C07306=1192.829,186.350,-57.414,-177.869,6.477,148.554
C07307=1192.833,186.102,-57.391,-177.872,6.475,148.554
C07308=1192.838,185.853,-57.368,-177.874,6.474,148.554
C07309=1192.842,185.604,-57.345,-177.877,6.472,148.555
C07310=1192.846,185.355,-57.322,-177.880,6.470,148.555
C07311=1192.852,185.085,-57.297,-177.883,6.467,148.555
C07312=1192.857,184.815,-57.272,-177.885,6.466,148.556
C07313=1192.862,184.546,-57.247,-177.888,6.464,148.556
C07314=1192.867,184.276,-57.222,-177.891,6.462,148.556
C07315=1192.872,184.027,-57.199,-177.893,6.460,148.557
C07316=1192.876,183.779,-57.177,-177.896,6.458,148.557
C07317=1192.881,183.530,-57.153,-177.899,6.457,148.558
C07318=1192.885,183.281,-57.131,-177.901,6.455,148.558
C07319=1192.890,183.032,-57.108,-177.904,6.453,148.558
C07320=1192.894,182.783,-57.084,-177.907,6.451,148.559
C07321=1192.899,182.535,-57.062,-177.909,6.449,148.559
C07322=1192.904,182.285,-57.039,-177.912,6.448,148.559
C07323=1192.908,182.036,-57.017,-177.915,6.446,148.560
C07324=1192.913,181.787,-56.993,-177.917,6.444,148.560
C07325=1192.918,181.538,-56.971,-177.920,6.442,148.560
C07326=1192.922,181.290,-56.948,-177.923,6.440,148.561
C07327=1192.927,181.040,-56.925,-177.925,6.439,148.561
C07328=1192.931,180.791,-56.903,-177.928,6.437,148.561
C07329=1192.937,180.543,-56.880,-177.931,6.435,148.562
C07330=1192.941,180.294,-56.857,-177.933,6.433,148.562
C07331=1192.946,180.044,-56.834,-177.936,6.431,148.563
C07332=1192.950,179.796,-56.812,-177.939,6.430,148.563
C07333=1192.955,179.547,-56.789,-177.941,6.428,148.563
C07334=1192.959,179.298,-56.767,-177.944,6.426,148.564
C07335=1192.964,179.049,-56.743,-177.947,6.424,148.564
C07336=1192.969,178.800,-56.722,-177.949,6.422,148.564
C07337=1192.973,178.551,-56.698,-177.952,6.421,148.565
C07338=1192.978,178.302,-56.676,-177.955,6.419,148.565
C07339=1192.983,178.054,-56.653,-177.957,6.417,148.565
C07340=1192.987,177.804,-56.631,-177.960,6.415,148.566
C07341=1192.992,177.555,-56.608,-177.962,6.414,148.566
C07342=1192.997,177.307,-56.586,-177.965,6.412,148.567
C07343=1193.001,177.058,-56.563,-177.968,6.411,148.567
C07344=1193.006,176.808,-56.541,-177.970,6.409,148.567
C07345=1193.010,176.560,-56.518,-177.973,6.407,148.568
C07346=1193.015,176.311,-56.496,-177.976,6.405,148.568
C07347=1193.019,176.062,-56.473,-177.978,6.403,148.568
C07348=1193.025,175.813,-56.451,-177.981,6.402,148.569
C07349=1193.029,175.564,-56.428,-177.984,6.400,148.569
C07350=1193.033,175.315,-56.406,-177.986,6.398,148.569
C07351=1193.039,175.066,-56.384,-177.989,6.396,148.570
C07352=1193.043,174.817,-56.361,-177.992,6.395,148.570
C07353=1193.048,174.569,-56.339,-177.994,6.393,148.570
C07354=1193.053,174.319,-56.316,-177.997,6.391,148.571
C07355=1193.056,174.070,-56.294,-178.000,6.389,148.571
C07356=1193.061,173.822,-56.272,-178.002,6.387,148.572
C07357=1193.066,173.573,-56.249,-178.004,6.386,148.572
C07358=1193.071,173.324,-56.227,-178.007,6.385,148.572
C07359=1193.075,173.075,-56.205,-178.010,6.383,148.573
C07360=1193.080,172.825,-56.182,-178.012,6.381,148.573
C07361=1193.085,172.577,-56.160,-178.016,6.380,148.574
C07362=1193.089,172.328,-56.138,-178.018,6.378,148.574
C07363=1193.095,172.079,-56.116,-178.021,6.376,148.574
C07364=1193.099,171.830,-56.093,-178.024,6.374,148.575
C07365=1193.103,171.581,-56.071,-178.026,6.372,148.575
C07366=1193.108,171.332,-56.048,-178.029,6.371,148.575
C07367=1193.113,171.082,-56.026,-178.032,6.369,148.576
C07368=1193.118,170.834,-56.005,-178.034,6.368,148.576
C07369=1193.122,170.585,-55.982,-178.036,6.366,148.577
C07370=1193.127,170.336,-55.960,-178.039,6.364,148.577
C07371=1193.131,170.087,-55.938,-178.042,6.362,148.577
C07372=1193.136,169.838,-55.916,-178.044,6.361,148.578
C07373=1193.141,169.589,-55.894,-178.047,6.359,148.578
C07374=1193.145,169.341,-55.872,-178.050,6.357,148.578
C07375=1193.150,169.091,-55.849,-178.052,6.355,148.579
C07376=1193.155,168.842,-55.827,-178.055,6.354,148.579
C07377=1193.159,168.593,-55.805,-178.058,6.352,148.579
C07378=1193.164,168.344,-55.783,-178.060,6.351,148.580
C07379=1193.168,168.095,-55.761,-178.063,6.349,148.580
C07380=1193.174,167.846,-55.739,-178.066,6.348,148.581
C07381=1193.178,167.597,-55.717,-178.068,6.346,148.581
C07382=1193.183,167.348,-55.695,-178.071,6.344,148.582
C07383=1193.187,167.099,-55.673,-178.074,6.342,148.582
C07384=1193.192,166.850,-55.652,-178.076,6.340,148.582
C07385=1193.196,166.601,-55.629,-178.079,6.339,148.583
C07386=1193.201,166.353,-55.607,-178.081,6.338,148.583
C07387=1193.206,166.103,-55.585,-178.084,6.336,148.583
C07388=1193.211,165.854,-55.563,-178.087,6.334,148.584
C07389=1193.215,165.605,-55.541,-178.089,6.332,148.584
C07390=1193.220,165.356,-55.519,-178.092,6.331,148.585
C07391=1193.225,165.108,-55.498,-178.095,6.329,148.585
C07392=1193.230,164.858,-55.476,-178.098,6.327,148.585
C07393=1193.234,164.609,-55.454,-178.100,6.326,148.586
C07394=1193.239,164.360,-55.432,-178.102,6.325,148.586
C07395=1193.244,164.111,-55.411,-178.105,6.323,148.587
C07396=1193.248,163.862,-55.389,-178.108,6.321,148.587
C07397=1193.253,163.613,-55.367,-178.111,6.319,148.587
C07398=1193.258,163.365,-55.345,-178.113,6.317,148.588
C07399=1193.262,163.115,-55.323,-178.116,6.316,148.588
C07400=1193.267,162.867,-55.302,-178.119,6.314,148.588
C07401=1193.271,162.617,-55.280,-178.121,6.313,148.589
C07402=1193.276,162.368,-55.259,-178.124,6.311,148.589
C07403=1193.281,162.119,-55.237,-178.126,6.310,148.590
C07404=1193.285,161.870,-55.215,-178.129,6.308,148.590
C07405=1193.290,161.621,-55.193,-178.132,6.306,148.591
C07406=1193.294,161.372,-55.171,-178.135,6.304,148.591
C07407=1193.299,161.123,-55.149,-178.137,6.303,148.591
C07408=1193.304,160.874,-55.128,-178.139,6.302,148.592
C07409=1193.309,160.625,-55.106,-178.142,6.300,148.592
C07410=1193.314,160.376,-55.085,-178.145,6.298,148.593
C07411=1193.319,160.128,-55.063,-178.148,6.297,148.593
C07412=1193.323,159.878,-55.042,-178.150,6.295,148.593
C07413=1193.328,159.629,-55.020,-178.153,6.294,148.594
C07414=1193.333,159.380,-54.998,-178.155,6.292,148.594
C07415=1193.338,159.111,-54.976,-178.158,6.290,148.595
C07416=1193.343,158.842,-54.952,-178.161,6.289,148.595
C07417=1193.347,158.573,-54.929,-178.164,6.287,148.596
C07418=1193.353,158.304,-54.905,-178.166,6.285,148.596
C07419=1193.357,158.055,-54.883,-178.169,6.283,148.596
C07420=1193.362,157.805,-54.862,-178.172,6.282,148.597
C07421=1193.367,157.557,-54.841,-178.175,6.280,148.597
C07422=1193.371,157.308,-54.819,-178.178,6.278,148.598
C07423=1193.376,157.059,-54.798,-178.180,6.277,148.598
C07424=1193.381,156.810,-54.777,-178.182,6.276,148.598
C07425=1193.386,156.561,-54.756,-178.185,6.274,148.599
C07426=1193.390,156.311,-54.734,-178.188,6.272,148.599
C07427=1193.395,156.063,-54.712,-178.191,6.271,148.600
C07428=1193.400,155.813,-54.691,-178.194,6.269,148.600
C07429=1193.404,155.565,-54.670,-178.196,6.268,148.600
C07430=1193.409,155.315,-54.649,-178.198,6.266,148.601
C07431=1193.414,155.066,-54.627,-178.201,6.264,148.601
C07432=1193.419,154.817,-54.606,-178.204,6.263,148.602
C07433=1193.423,154.568,-54.584,-178.206,6.261,148.602
C07434=1193.428,154.319,-54.563,-178.209,6.260,148.603
C07435=1193.433,154.070,-54.542,-178.212,6.258,148.603
C07436=1193.438,153.821,-54.521,-178.214,6.257,148.603
C07437=1193.443,153.572,-54.499,-178.217,6.255,148.604
C07438=1193.447,153.323,-54.478,-178.219,6.254,148.604
C07439=1193.451,153.074,-54.457,-178.222,6.252,148.604
C07440=1193.457,152.825,-54.436,-178.225,6.251,148.605
C07441=1193.461,152.576,-54.414,-178.228,6.249,148.605
C07442=1193.465,152.327,-54.393,-178.230,6.247,148.606
C07443=1193.470,152.078,-54.372,-178.233,6.246,148.606
C07444=1193.475,151.829,-54.351,-178.235,6.244,148.607
C07445=1193.480,151.580,-54.330,-178.238,6.243,148.607
C07446=1193.485,151.331,-54.309,-178.241,6.241,148.608
C07447=1193.489,151.081,-54.287,-178.243,6.240,148.608
C07448=1193.494,150.832,-54.267,-178.246,6.239,148.608
C07449=1193.499,150.583,-54.245,-178.249,6.237,148.609
C07450=1193.504,150.334,-54.224,-178.251,6.235,148.609
C07451=1193.508,150.085,-54.204,-178.254,6.234,148.610
C07452=1193.513,149.837,-54.182,-178.256,6.233,148.610
C07453=1193.518,149.587,-54.161,-178.259,6.231,148.610
C07454=1193.522,149.338,-54.141,-178.262,6.229,148.611
C07455=1193.527,149.089,-54.119,-178.265,6.227,148.611
C07456=1193.532,148.840,-54.098,-178.267,6.227,148.612
C07457=1193.537,148.591,-54.077,-178.270,6.225,148.612
C07458=1193.542,148.342,-54.057,-178.273,6.223,148.613
C07459=1193.546,148.093,-54.035,-178.275,6.221,148.613
C07460=1193.550,147.843,-54.014,-178.277,6.220,148.613
C07461=1193.556,147.594,-53.993,-178.280,6.219,148.614
C07462=1193.560,147.345,-53.973,-178.283,6.217,148.614
C07463=1193.565,147.096,-53.951,-178.286,6.215,148.615
C07464=1193.569,146.848,-53.931,-178.288,6.214,148.615
C07465=1193.574,146.598,-53.910,-178.291,6.213,148.616
C07466=1193.579,146.349,-53.889,-178.294,6.211,148.616
C07467=1193.584,146.100,-53.868,-178.296,6.209,148.617
C07468=1193.589,145.851,-53.847,-178.299,6.209,148.617
C07469=1193.593,145.602,-53.826,-178.301,6.207,148.617
C07470=1193.598,145.353,-53.805,-178.304,6.205,148.618
C07471=1193.602,145.104,-53.785,-178.307,6.204,148.618
C07472=1193.608,144.854,-53.764,-178.309,6.203,148.619
C07473=1193.612,144.605,-53.743,-178.312,6.201,148.619
C07474=1193.617,144.356,-53.722,-178.315,6.199,148.619
C07475=1193.622,144.107,-53.702,-178.317,6.198,148.620
C07476=1193.627,143.858,-53.681,-178.320,6.197,148.620
C07477=1193.631,143.609,-53.661,-178.323,6.195,148.621
C07478=1193.636,143.360,-53.640,-178.325,6.193,148.621
C07479=1193.641,143.111,-53.619,-178.328,6.193,148.622
C07480=1193.645,142.862,-53.598,-178.331,6.191,148.622
C07481=1193.650,142.613,-53.577,-178.333,6.189,148.623
C07482=1193.655,142.364,-53.557,-178.335,6.188,148.623
C07483=1193.660,142.115,-53.536,-178.338,6.186,148.623
C07484=1193.664,141.866,-53.516,-178.341,6.185,148.624
C07485=1193.669,141.617,-53.495,-178.344,6.183,148.624
C07486=1193.674,141.368,-53.474,-178.346,6.182,148.625
C07487=1193.679,141.118,-53.455,-178.349,6.180,148.625
C07488=1193.684,140.869,-53.434,-178.352,6.179,148.626
C07489=1193.688,140.620,-53.413,-178.354,6.178,148.626
C07490=1193.693,140.371,-53.393,-178.357,6.176,148.627
C07491=1193.698,140.122,-53.372,-178.359,6.174,148.627
C07492=1193.702,139.873,-53.351,-178.362,6.174,148.628
C07493=1193.707,139.624,-53.331,-178.365,6.172,148.628
C07494=1193.712,139.375,-53.310,-178.367,6.170,148.628
C07495=1193.716,139.126,-53.290,-178.370,6.169,148.629
C07496=1193.721,138.876,-53.269,-178.373,6.168,148.629
C07497=1193.726,138.627,-53.248,-178.375,6.166,148.630
C07498=1193.731,138.378,-53.229,-178.378,6.164,148.630
C07499=1193.736,138.129,-53.208,-178.381,6.164,148.631
C07500=1193.740,137.880,-53.187,-178.383,6.162,148.631
C07501=1193.745,137.631,-53.167,-178.386,6.160,148.632
C07502=1193.749,137.382,-53.147,-178.388,6.159,148.632
C07503=1193.755,137.132,-53.126,-178.391,6.158,148.633
C07504=1193.759,136.883,-53.106,-178.394,6.156,148.633
C07505=1193.763,136.634,-53.086,-178.396,6.155,148.633
C07506=1193.769,136.385,-53.065,-178.399,6.153,148.634
C07507=1193.773,136.135,-53.045,-178.402,6.152,148.634
C07508=1193.778,135.886,-53.025,-178.404,6.151,148.635
C07509=1193.782,135.637,-53.004,-178.407,6.149,148.635
C07510=1193.788,135.389,-52.984,-178.410,6.148,148.636
C07511=1193.793,135.139,-52.964,-178.412,6.147,148.636
C07512=1193.797,134.890,-52.944,-178.415,6.145,148.637
C07513=1193.802,134.641,-52.923,-178.417,6.143,148.637
C07514=1193.806,134.392,-52.904,-178.420,6.143,148.638
C07515=1193.812,134.142,-52.883,-178.423,6.141,148.638
C07516=1193.816,133.893,-52.862,-178.425,6.139,148.638
C07517=1193.821,133.644,-52.843,-178.428,6.139,148.639
C07518=1193.825,133.395,-52.822,-178.431,6.137,148.639
C07519=1193.831,133.127,-52.800,-178.433,6.135,148.640
C07520=1193.835,132.858,-52.779,-178.437,6.134,148.640
C07521=1193.841,132.589,-52.757,-178.439,6.132,148.641
C07522=1193.846,132.321,-52.735,-178.442,6.131,148.641
C07523=1193.851,132.071,-52.715,-178.445,6.130,148.642
C07524=1193.856,131.823,-52.695,-178.447,6.128,148.642
C07525=1193.861,131.573,-52.675,-178.450,6.127,148.643
C07526=1193.865,131.324,-52.655,-178.453,6.125,148.643
C07527=1193.870,131.075,-52.635,-178.455,6.124,148.644
C07528=1193.875,130.826,-52.615,-178.458,6.123,148.644
C07529=1193.879,130.577,-52.595,-178.461,6.121,148.645
C07530=1193.884,130.328,-52.575,-178.463,6.120,148.645
C07531=1193.890,130.079,-52.554,-178.465,6.119,148.645
C07532=1193.894,129.829,-52.535,-178.469,6.117,148.646
C07533=1193.899,129.580,-52.514,-178.471,6.115,148.646
C07534=1193.903,129.331,-52.495,-178.473,6.114,148.647
C07535=1193.909,129.082,-52.475,-178.476,6.113,148.647
C07536=1193.913,128.833,-52.455,-178.479,6.112,148.648
C07537=1193.918,128.583,-52.435,-178.481,6.110,148.648
C07538=1193.922,128.334,-52.415,-178.484,6.109,148.649
C07539=1193.927,128.085,-52.395,-178.487,6.108,148.649
C07540=1193.932,127.837,-52.375,-178.489,6.106,148.650
C07541=1193.937,127.587,-52.356,-178.492,6.106,148.650
C07542=1193.941,127.338,-52.335,-178.495,6.104,148.651
C07543=1193.946,127.088,-52.316,-178.497,6.102,148.651
C07544=1193.951,126.840,-52.296,-178.500,6.102,148.652
C07545=1193.956,126.591,-52.276,-178.503,6.100,148.652
C07546=1193.961,126.341,-52.256,-178.505,6.098,148.652
C07547=1193.965,126.091,-52.237,-178.508,6.097,148.653
C07548=1193.970,125.843,-52.217,-178.511,6.096,148.653
C07549=1193.975,125.594,-52.197,-178.513,6.095,148.654
C07550=1193.980,125.344,-52.177,-178.516,6.093,148.654
C07551=1193.984,125.095,-52.157,-178.519,6.092,148.655
C07552=1193.990,124.846,-52.138,-178.521,6.091,148.655
C07553=1193.994,124.597,-52.118,-178.524,6.089,148.656
C07554=1193.999,124.347,-52.098,-178.526,6.088,148.656
C07555=1194.004,124.098,-52.078,-178.529,6.087,148.657
C07556=1194.009,123.849,-52.059,-178.532,6.085,148.657
C07557=1194.013,123.600,-52.040,-178.534,6.084,148.658
C07558=1194.018,123.350,-52.020,-178.537,6.082,148.658
C07559=1194.023,123.102,-52.000,-178.539,6.082,148.659
C07560=1194.028,122.853,-51.980,-178.542,6.080,148.659
C07561=1194.032,122.603,-51.961,-178.544,6.079,148.660
C07562=1194.038,122.354,-51.941,-178.547,6.078,148.660
C07563=1194.042,122.105,-51.921,-178.550,6.076,148.661
C07564=1194.047,121.856,-51.901,-178.553,6.075,148.661
C07565=1194.052,121.607,-51.882,-178.555,6.074,148.662
C07566=1194.056,121.358,-51.863,-178.557,6.073,148.662
C07567=1194.061,121.108,-51.843,-178.561,6.071,148.663
C07568=1194.066,120.859,-51.824,-178.563,6.070,148.663
C07569=1194.071,120.610,-51.804,-178.565,6.069,148.663
C07570=1194.075,120.361,-51.784,-178.569,6.067,148.664
C07571=1194.081,120.112,-51.765,-178.571,6.066,148.664
C07572=1194.085,119.863,-51.746,-178.573,6.064,148.665
C07573=1194.089,119.613,-51.726,-178.576,6.064,148.666
C07574=1194.095,119.364,-51.707,-178.579,6.062,148.666
C07575=1194.100,119.115,-51.687,-178.582,6.061,148.667
C07576=1194.105,118.866,-51.668,-178.584,6.060,148.667
C07577=1194.109,118.616,-51.649,-178.587,6.058,148.667
C07578=1194.114,118.367,-51.629,-178.589,6.057,148.668
C07579=1194.119,118.118,-51.610,-178.592,6.056,148.668
C07580=1194.124,117.868,-51.590,-178.594,6.055,148.669
C07581=1194.128,117.620,-51.571,-178.597,6.053,148.669
C07582=1194.133,117.370,-51.552,-178.599,6.052,148.670
C07583=1194.138,117.121,-51.532,-178.603,6.051,148.670
C07584=1194.143,116.872,-51.513,-178.605,6.049,148.671
C07585=1194.147,116.623,-51.494,-178.607,6.048,148.671
C07586=1194.153,116.374,-51.475,-178.611,6.047,148.672
C07587=1194.157,116.124,-51.455,-178.613,6.046,148.672
C07588=1194.162,115.876,-51.436,-178.616,6.045,148.673
C07589=1194.167,115.626,-51.416,-178.618,6.044,148.673
C07590=1194.172,115.377,-51.397,-178.621,6.042,148.674
C07591=1194.177,115.128,-51.378,-178.623,6.041,148.674
C07592=1194.181,114.878,-51.358,-178.626,6.040,148.675
C07593=1194.186,114.629,-51.340,-178.629,6.039,148.675
C07594=1194.191,114.379,-51.320,-178.631,6.037,148.676
C07595=1194.196,114.131,-51.302,-178.634,6.036,148.676
C07596=1194.200,113.881,-51.282,-178.637,6.035,148.677
C07597=1194.206,113.632,-51.263,-178.639,6.034,148.677
C07598=1194.210,113.383,-51.244,-178.642,6.033,148.678
C07599=1194.215,113.134,-51.224,-178.645,6.031,148.678
C07600=1194.219,112.884,-51.206,-178.647,6.030,148.679
C07601=1194.225,112.635,-51.187,-178.650,6.029,148.679
C07602=1194.230,112.386,-51.167,-178.652,6.028,148.680
C07603=1194.234,112.137,-51.148,-178.655,6.026,148.680
C07604=1194.239,111.888,-51.129,-178.658,6.025,148.681
C07605=1194.244,111.639,-51.111,-178.660,6.023,148.681
C07606=1194.249,111.389,-51.091,-178.663,6.023,148.682
C07607=1194.254,111.140,-51.072,-178.666,6.021,148.682
C07608=1194.258,110.891,-51.053,-178.668,6.021,148.683
C07609=1194.264,110.641,-51.034,-178.671,6.019,148.683
C07610=1194.268,110.392,-51.015,-178.673,6.018,148.684
C07611=1194.273,110.143,-50.996,-178.676,6.017,148.684
C07612=1194.277,109.893,-50.977,-178.678,6.016,148.685
C07613=1194.283,109.645,-50.958,-178.681,6.014,148.685
C07614=1194.287,109.396,-50.939,-178.684,6.013,148.686
C07615=1194.292,109.146,-50.920,-178.687,6.012,148.686
C07616=1194.297,108.897,-50.902,-178.689,6.011,148.687
C07617=1194.302,108.648,-50.882,-178.692,6.010,148.687
C07618=1194.306,108.398,-50.864,-178.694,6.009,148.688
C07619=1194.311,108.149,-50.844,-178.697,6.007,148.688
C07620=1194.316,107.900,-50.826,-178.700,6.006,148.689
C07621=1194.321,107.650,-50.807,-178.702,6.005,148.689
C07622=1194.325,107.402,-50.788,-178.705,6.004,148.690
C07623=1194.331,107.133,-50.768,-178.708,6.002,148.690
C07624=1194.336,106.864,-50.747,-178.711,6.001,148.691
C07625=1194.341,106.596,-50.728,-178.713,6.000,148.692
C07626=1194.347,106.328,-50.707,-178.716,5.998,148.692
C07627=1194.351,106.078,-50.689,-178.719,5.998,148.693
C07628=1194.356,105.829,-50.669,-178.721,5.996,148.693
C07629=1194.361,105.580,-50.651,-178.724,5.996,148.694
C07630=1194.366,105.331,-50.632,-178.727,5.994,148.694
C07631=1194.371,105.082,-50.614,-178.729,5.993,148.695
C07632=1194.376,104.832,-50.594,-178.732,5.992,148.695
C07633=1194.381,104.583,-50.576,-178.734,5.991,148.696
C07634=1194.385,104.334,-50.557,-178.737,5.989,148.696
C07635=1194.390,104.084,-50.538,-178.739,5.988,148.697
C07636=1194.395,103.835,-50.520,-178.743,5.987,148.697
C07637=1194.400,103.586,-50.502,-178.745,5.986,148.698
C07638=1194.405,103.337,-50.482,-178.748,5.985,148.698
C07639=1194.410,103.088,-50.464,-178.750,5.984,148.699
C07640=1194.415,102.839,-50.445,-178.753,5.983,148.699
C07641=1194.419,102.589,-50.426,-178.755,5.981,148.700
C07642=1194.424,102.340,-50.408,-178.758,5.980,148.700
C07643=1194.429,102.091,-50.389,-178.761,5.979,148.701
C07644=1194.434,101.841,-50.371,-178.763,5.978,148.701
C07645=1194.438,101.592,-50.352,-178.766,5.977,148.702
C07646=1194.444,101.343,-50.334,-178.768,5.976,148.702
C07647=1194.448,101.093,-50.315,-178.771,5.974,148.703
C07648=1194.453,100.844,-50.296,-178.774,5.973,148.703
C07649=1194.458,100.595,-50.279,-178.777,5.972,148.704
C07650=1194.463,100.345,-50.260,-178.779,5.971,148.704
C07651=1194.467,100.096,-50.241,-178.781,5.971,148.705
C07652=1194.472,99.847,-50.223,-178.784,5.969,148.706
C07653=1194.477,99.597,-50.204,-178.787,5.968,148.706
C07654=1194.482,99.349,-50.185,-178.790,5.967,148.707
C07655=1194.487,99.099,-50.167,-178.792,5.966,148.707
C07656=1194.492,98.850,-50.149,-178.795,5.964,148.708
C07657=1194.497,98.600,-50.130,-178.797,5.964,148.708
C07658=1194.502,98.351,-50.112,-178.800,5.963,148.709
C07659=1194.506,98.102,-50.094,-178.803,5.961,148.709
C07660=1194.511,97.853,-50.076,-178.805,5.960,148.710
C07661=1194.516,97.603,-50.057,-178.808,5.959,148.710
C07662=1194.521,97.354,-50.039,-178.810,5.958,148.711
C07663=1194.526,97.105,-50.020,-178.813,5.957,148.711
C07664=1194.531,96.856,-50.002,-178.816,5.956,148.712
C07665=1194.535,96.606,-49.984,-178.818,5.955,148.713
C07666=1194.540,96.357,-49.966,-178.821,5.953,148.713
C07667=1194.546,96.107,-49.947,-178.824,5.953,148.714
C07668=1194.550,95.859,-49.929,-178.826,5.951,148.714
C07669=1194.555,95.610,-49.911,-178.829,5.951,148.715
C07670=1194.560,95.360,-49.892,-178.832,5.949,148.715
C07671=1194.564,95.111,-49.874,-178.834,5.948,148.716
C07672=1194.569,94.862,-49.856,-178.836,5.947,148.716
C07673=1194.574,94.612,-49.838,-178.840,5.946,148.717
C07674=1194.580,94.363,-49.820,-178.842,5.945,148.717
C07675=1194.584,94.113,-49.801,-178.845,5.944,148.718
C07676=1194.589,93.864,-49.783,-178.847,5.943,148.718
C07677=1194.594,93.615,-49.765,-178.850,5.942,148.719
C07678=1194.599,93.366,-49.747,-178.852,5.940,148.719
C07679=1194.604,93.117,-49.729,-178.855,5.940,148.720
C07680=1194.608,92.867,-49.710,-178.858,5.938,148.720
C07681=1194.613,92.618,-49.692,-178.860,5.938,148.721
C07682=1194.618,92.369,-49.674,-178.862,5.937,148.721
C07683=1194.623,92.120,-49.656,-178.866,5.935,148.722
C07684=1194.628,91.870,-49.638,-178.868,5.934,148.722
C07685=1194.633,91.621,-49.620,-178.871,5.933,148.723
C07686=1194.638,91.372,-49.602,-178.873,5.932,148.724
C07687=1194.642,91.122,-49.584,-178.876,5.932,148.724
C07688=1194.647,90.873,-49.566,-178.878,5.930,148.725
C07689=1194.652,90.623,-49.548,-178.881,5.929,148.725
C07690=1194.657,90.374,-49.530,-178.884,5.928,148.726
C07691=1194.662,90.125,-49.512,-178.886,5.927,148.726
C07692=1194.667,89.875,-49.494,-178.888,5.926,148.727
C07693=1194.672,89.626,-49.476,-178.892,5.925,148.727
C07694=1194.677,89.377,-49.458,-178.894,5.924,148.728
C07695=1194.681,89.127,-49.440,-178.896,5.923,148.728
C07696=1194.686,88.878,-49.422,-178.899,5.921,148.729
C07697=1194.691,88.629,-49.404,-178.902,5.921,148.730
C07698=1194.696,88.380,-49.386,-178.904,5.919,148.730
C07699=1194.701,88.130,-49.368,-178.907,5.919,148.731
C07700=1194.706,87.881,-49.350,-178.910,5.918,148.731
C07701=1194.711,87.631,-49.333,-178.912,5.916,148.732
C07702=1194.715,87.383,-49.315,-178.915,5.916,148.732
C07703=1194.720,87.133,-49.298,-178.917,5.915,148.733
C07704=1194.725,86.884,-49.280,-178.920,5.913,148.733
C07705=1194.730,86.635,-49.262,-178.923,5.913,148.734
C07706=1194.735,86.385,-49.244,-178.925,5.912,148.734
C07707=1194.740,86.136,-49.226,-178.928,5.910,148.735
C07708=1194.745,85.886,-49.208,-178.930,5.910,148.736
C07709=1194.749,85.637,-49.190,-178.933,5.908,148.736
C07710=1194.754,85.388,-49.172,-178.936,5.907,148.737
C07711=1194.760,85.138,-49.155,-178.938,5.907,148.737
C07712=1194.764,84.889,-49.137,-178.941,5.905,148.738
C07713=1194.769,84.640,-49.119,-178.944,5.905,148.738
C07714=1194.774,84.391,-49.101,-178.946,5.904,148.739
C07715=1194.779,84.141,-49.084,-178.949,5.902,148.739
C07716=1194.784,83.892,-49.066,-178.951,5.901,148.740
C07717=1194.789,83.643,-49.048,-178.954,5.901,148.740
C07718=1194.794,83.393,-49.031,-178.957,5.899,148.741
C07719=1194.799,83.144,-49.013,-178.959,5.898,148.742
C07720=1194.803,82.895,-48.996,-178.961,5.898,148.742
C07721=1194.808,82.645,-48.978,-178.965,5.896,148.743
C07722=1194.813,82.396,-48.960,-178.967,5.896,148.743
C07723=1194.818,82.147,-48.942,-178.969,5.895,148.744
C07724=1194.823,81.897,-48.925,-178.973,5.893,148.744
C07725=1194.827,81.648,-48.908,-178.975,5.892,148.745
C07726=1194.833,81.398,-48.890,-178.977,5.892,148.745
C07727=1194.838,81.130,-48.871,-178.980,5.891,148.746
C07728=1194.844,80.862,-48.853,-178.983,5.890,148.747
C07729=1194.849,80.594,-48.833,-178.986,5.888,148.747
C07730=1194.854,80.325,-48.815,-178.988,5.888,148.748
C07731=1194.858,80.076,-48.797,-178.991,5.886,148.748
C07732=1194.863,79.826,-48.780,-178.994,5.885,148.749
C07733=1194.868,79.577,-48.762,-178.996,5.885,148.750
C07734=1194.873,79.328,-48.744,-178.999,5.883,148.750
C07735=1194.878,79.078,-48.727,-179.002,5.883,148.751
C07736=1194.883,78.829,-48.709,-179.004,5.882,148.751
C07737=1194.889,78.580,-48.692,-179.007,5.880,148.752
C07738=1194.893,78.331,-48.674,-179.010,5.880,148.752
C07739=1194.898,78.081,-48.658,-179.012,5.879,148.753
C07740=1194.903,77.832,-48.640,-179.015,5.877,148.753
C07741=1194.908,77.582,-48.623,-179.017,5.877,148.754
C07742=1194.913,77.333,-48.606,-179.020,5.876,148.755
C07743=1194.917,77.084,-48.588,-179.022,5.875,148.755
C07744=1194.923,76.834,-48.571,-179.025,5.874,148.756
C07745=1194.927,76.585,-48.553,-179.028,5.873,148.756
C07746=1194.932,76.335,-48.536,-179.030,5.872,148.757
C07747=1194.937,76.086,-48.518,-179.033,5.871,148.757
C07748=1194.942,75.837,-48.502,-179.035,5.870,148.758
C07749=1194.947,75.587,-48.484,-179.038,5.869,148.758
C07750=1194.952,75.338,-48.466,-179.041,5.868,148.759
C07751=1194.957,75.089,-48.450,-179.043,5.867,148.760
C07752=1194.962,74.840,-48.432,-179.046,5.867,148.760
C07753=1194.966,74.590,-48.415,-179.048,5.866,148.761
C07754=1194.971,74.340,-48.398,-179.051,5.864,148.761
C07755=1194.977,74.092,-48.380,-179.053,5.863,148.762
C07756=1194.981,73.842,-48.364,-179.056,5.863,148.762
C07757=1194.986,73.593,-48.346,-179.059,5.862,148.763
C07758=1194.991,73.344,-48.329,-179.061,5.861,148.763
C07759=1194.996,73.094,-48.312,-179.064,5.860,148.764
C07760=1195.000,72.844,-48.295,-179.066,5.859,148.765
C07761=1195.006,72.595,-48.278,-179.069,5.858,148.765
C07762=1195.011,72.346,-48.260,-179.072,5.857,148.766
C07763=1195.016,72.097,-48.243,-179.074,5.856,148.766
C07764=1195.021,71.847,-48.226,-179.077,5.855,148.767
C07765=1195.025,71.597,-48.209,-179.080,5.854,148.768
C07766=1195.030,71.348,-48.192,-179.082,5.854,148.768
C07767=1195.035,71.099,-48.175,-179.085,5.853,148.769
C07768=1195.040,70.850,-48.158,-179.087,5.851,148.769
C07769=1195.045,70.600,-48.141,-179.090,5.851,148.770
C07770=1195.050,70.351,-48.123,-179.093,5.850,148.770
C07771=1195.054,70.101,-48.107,-179.095,5.849,148.771
C07772=1195.060,69.852,-48.090,-179.098,5.848,148.772
C07773=1195.065,69.603,-48.073,-179.100,5.847,148.772
C07774=1195.070,69.353,-48.056,-179.103,5.846,148.773
C07775=1195.074,69.104,-48.039,-179.105,5.846,148.773
C07776=1195.080,68.855,-48.022,-179.108,5.844,148.774
C07777=1195.084,68.606,-48.005,-179.111,5.844,148.774
C07778=1195.090,68.356,-47.988,-179.113,5.843,148.775
C07779=1195.094,68.106,-47.971,-179.116,5.842,148.775
C07780=1195.100,67.857,-47.954,-179.119,5.841,148.776
C07781=1195.104,67.608,-47.937,-179.121,5.840,148.777
C07782=1195.109,67.358,-47.921,-179.124,5.839,148.777
C07783=1195.114,67.108,-47.903,-179.126,5.839,148.778
C07784=1195.119,66.860,-47.887,-179.129,5.837,148.778
C07785=1195.124,66.611,-47.869,-179.132,5.837,148.779
C07786=1195.128,66.361,-47.852,-179.134,5.836,148.779
C07787=1195.133,66.112,-47.836,-179.136,5.835,148.780
C07788=1195.139,65.862,-47.819,-179.140,5.834,148.781
C07789=1195.143,65.613,-47.802,-179.142,5.833,148.781
C07790=1195.148,65.363,-47.785,-179.144,5.832,148.782
C07791=1195.154,65.114,-47.769,-179.147,5.832,148.782
C07792=1195.158,64.865,-47.752,-179.150,5.830,148.783
C07793=1195.163,64.615,-47.735,-179.152,5.830,148.784
C07794=1195.168,64.366,-47.718,-179.155,5.829,148.784
C07795=1195.173,64.117,-47.702,-179.157,5.828,148.785
C07796=1195.178,63.867,-47.684,-179.160,5.827,148.785
C07797=1195.183,63.618,-47.668,-179.162,5.826,148.786
C07798=1195.188,63.369,-47.652,-179.165,5.825,148.786
C07799=1195.193,63.118,-47.635,-179.168,5.825,148.787
C07800=1195.198,62.869,-47.618,-179.170,5.824,148.788
C07801=1195.203,62.620,-47.602,-179.173,5.822,148.788
C07802=1195.208,62.370,-47.585,-179.176,5.822,148.789
C07803=1195.212,62.121,-47.568,-179.178,5.821,148.789
C07804=1195.217,61.872,-47.552,-179.180,5.821,148.790
C07805=1195.222,61.623,-47.535,-179.184,5.819,148.791
C07806=1195.227,61.373,-47.518,-179.186,5.818,148.791
C07807=1195.232,61.124,-47.502,-179.188,5.818,148.792
C07808=1195.237,60.875,-47.485,-179.191,5.817,148.792
C07809=1195.243,60.625,-47.469,-179.193,5.816,148.793
C07810=1195.247,60.375,-47.452,-179.196,5.815,148.793
C07811=1195.252,60.126,-47.435,-179.199,5.814,148.794
C07812=1195.257,59.877,-47.419,-179.201,5.813,148.795
C07813=1195.262,59.627,-47.402,-179.204,5.813,148.795
C07814=1195.267,59.377,-47.386,-179.206,5.812,148.796
C07815=1195.272,59.128,-47.369,-179.209,5.811,148.796
C07816=1195.276,58.879,-47.353,-179.212,5.810,148.797
C07817=1195.282,58.630,-47.337,-179.214,5.809,148.797
C07818=1195.287,58.380,-47.319,-179.217,5.809,148.798
C07819=1195.292,58.130,-47.303,-179.219,5.808,148.799
C07820=1195.297,57.881,-47.287,-179.222,5.806,148.799
C07821=1195.301,57.632,-47.270,-179.225,5.806,148.800
C07822=1195.306,57.383,-47.254,-179.227,5.805,148.801
C07823=1195.312,57.133,-47.237,-179.229,5.805,148.801
C07824=1195.317,56.884,-47.221,-179.232,5.804,148.802
C07825=1195.321,56.634,-47.205,-179.235,5.803,148.802
C07826=1195.326,56.384,-47.189,-179.237,5.802,148.803
C07827=1195.331,56.136,-47.172,-179.240,5.801,148.803
C07828=1195.336,55.886,-47.156,-179.243,5.801,148.804
C07829=1195.341,55.637,-47.140,-179.245,5.800,148.804
C07830=1195.346,55.387,-47.123,-179.247,5.799,148.805
C07831=1195.351,55.119,-47.105,-179.251,5.798,148.806
C07832=1195.357,54.851,-47.088,-179.253,5.797,148.806
C07833=1195.362,54.581,-47.071,-179.256,5.797,148.807
C07834=1195.367,54.314,-47.053,-179.259,5.795,148.808
C07835=1195.372,54.063,-47.037,-179.261,5.795,148.808
C07836=1195.378,53.814,-47.020,-179.264,5.794,148.809
C07837=1195.382,53.565,-47.003,-179.267,5.794,148.810
C07838=1195.388,53.315,-46.988,-179.269,5.793,148.810
C07839=1195.392,53.066,-46.971,-179.272,5.791,148.811
C07840=1195.398,52.817,-46.955,-179.275,5.791,148.811
C07841=1195.402,52.567,-46.939,-179.277,5.790,148.812
C07842=1195.407,52.318,-46.923,-179.279,5.789,148.812
C07843=1195.412,52.068,-46.907,-179.282,5.789,148.813
C07844=1195.417,51.819,-46.890,-179.284,5.788,148.814
C07845=1195.422,51.569,-46.874,-179.287,5.787,148.814
C07846=1195.427,51.321,-46.858,-179.290,5.786,148.815
C07847=1195.432,51.070,-46.842,-179.292,5.785,148.815
C07848=1195.437,50.822,-46.826,-179.295,5.785,148.816
C07849=1195.442,50.572,-46.810,-179.297,5.784,148.817
C07850=1195.447,50.323,-46.793,-179.300,5.783,148.817
C07851=1195.451,50.073,-46.778,-179.303,5.782,148.818
C07852=1195.456,49.824,-46.761,-179.305,5.781,148.818
C07853=1195.462,49.574,-46.746,-179.308,5.780,148.819
C07854=1195.467,49.324,-46.730,-179.310,5.780,148.820
C07855=1195.472,49.076,-46.713,-179.313,5.779,148.820
C07856=1195.477,48.825,-46.697,-179.316,5.779,148.821
C07857=1195.482,48.577,-46.681,-179.318,5.778,148.821
C07858=1195.486,48.327,-46.665,-179.321,5.777,148.822
C07859=1195.491,48.078,-46.649,-179.324,5.776,148.823
C07860=1195.496,47.828,-46.633,-179.326,5.775,148.823
C07861=1195.502,47.578,-46.617,-179.328,5.775,148.824
C07862=1195.507,47.330,-46.601,-179.331,5.774,148.824
C07863=1195.512,47.079,-46.585,-179.333,5.773,148.825
C07864=1195.516,46.830,-46.570,-179.336,5.773,148.826
C07865=1195.521,46.581,-46.553,-179.339,5.771,148.826
C07866=1195.526,46.331,-46.538,-179.341,5.770,148.827
C07867=1195.531,46.082,-46.522,-179.344,5.770,148.827
C07868=1195.536,45.833,-46.506,-179.346,5.769,148.828
C07869=1195.541,45.583,-46.490,-179.349,5.769,148.829
C07870=1195.546,45.333,-46.474,-179.351,5.768,148.829
C07871=1195.551,45.084,-46.458,-179.354,5.767,148.830
C07872=1195.557,44.835,-46.442,-179.356,5.767,148.830
C07873=1195.561,44.585,-46.427,-179.359,5.765,148.831
C07874=1195.566,44.336,-46.410,-179.362,5.765,148.832
C07875=1195.571,44.087,-46.395,-179.364,5.764,148.832
C07876=1195.576,43.837,-46.379,-179.367,5.763,148.833
C07877=1195.581,43.587,-46.363,-179.369,5.763,148.833
C07878=1195.586,43.338,-46.347,-179.372,5.762,148.834
C07879=1195.590,43.089,-46.332,-179.375,5.762,148.835
C07880=1195.596,42.839,-46.316,-179.377,5.761,148.835
C07881=1195.601,42.589,-46.300,-179.379,5.760,148.836
C07882=1195.606,42.340,-46.285,-179.383,5.759,148.837
C07883=1195.611,42.091,-46.268,-179.385,5.758,148.837
C07884=1195.616,41.841,-46.252,-179.387,5.758,148.838
C07885=1195.620,41.592,-46.237,-179.390,5.757,148.838
C07886=1195.626,41.342,-46.222,-179.393,5.757,148.839
C07887=1195.631,41.093,-46.206,-179.395,5.756,148.839
C07888=1195.636,40.843,-46.190,-179.397,5.755,148.840
C07889=1195.640,40.595,-46.174,-179.400,5.755,148.841
C07890=1195.646,40.345,-46.159,-179.402,5.754,148.841
C07891=1195.650,40.095,-46.143,-179.405,5.753,148.842
C07892=1195.656,39.846,-46.127,-179.408,5.752,148.843
C07893=1195.661,39.597,-46.112,-179.411,5.751,148.843
C07894=1195.665,39.346,-46.096,-179.413,5.750,148.844
C07895=1195.671,39.097,-46.081,-179.416,5.750,148.844
C07896=1195.676,38.848,-46.065,-179.418,5.749,148.845
C07897=1195.681,38.599,-46.050,-179.420,5.749,148.845
C07898=1195.686,38.348,-46.034,-179.423,5.748,148.846
C07899=1195.691,38.099,-46.019,-179.426,5.748,148.847
C07900=1195.696,37.850,-46.002,-179.428,5.747,148.847
C07901=1195.701,37.601,-45.987,-179.430,5.746,148.848
C07902=1195.705,37.351,-45.971,-179.433,5.746,148.849
C07903=1195.711,37.102,-45.956,-179.436,5.744,148.849
C07904=1195.715,36.853,-45.941,-179.439,5.744,148.850
C07905=1195.721,36.603,-45.925,-179.441,5.743,148.850
C07906=1195.726,36.353,-45.909,-179.444,5.742,148.851
C07907=1195.730,36.104,-45.894,-179.446,5.742,148.852
C07908=1195.736,35.855,-45.879,-179.448,5.741,148.852
C07909=1195.741,35.605,-45.863,-179.451,5.740,148.853
C07910=1195.745,35.355,-45.849,-179.454,5.740,148.854
C07911=1195.751,35.105,-45.833,-179.456,5.739,148.854
C07912=1195.755,34.856,-45.818,-179.459,5.738,148.855
C07913=1195.761,34.607,-45.802,-179.461,5.738,148.855
C07914=1195.766,34.357,-45.787,-179.464,5.737,148.856
C07915=1195.770,34.108,-45.771,-179.466,5.737,148.857
C07916=1195.776,33.858,-45.756,-179.469,5.736,148.857
C07917=1195.781,33.609,-45.740,-179.472,5.735,148.858
C07918=1195.786,33.360,-45.725,-179.475,5.734,148.858
C07919=1195.791,33.110,-45.710,-179.477,5.734,148.859
C07920=1195.795,32.861,-45.694,-179.479,5.733,148.860
C07921=1195.801,32.611,-45.679,-179.482,5.732,148.860
C07922=1195.805,32.361,-45.664,-179.485,5.732,148.861
C07923=1195.811,32.112,-45.649,-179.487,5.731,148.861
C07924=1195.816,31.863,-45.633,-179.489,5.730,148.862
C07925=1195.820,31.613,-45.618,-179.492,5.730,148.863
C07926=1195.826,31.363,-45.602,-179.495,5.729,148.863
C07927=1195.831,31.114,-45.588,-179.497,5.728,148.864
C07928=1195.836,30.864,-45.572,-179.499,5.728,148.865
C07929=1195.841,30.615,-45.557,-179.502,5.727,148.865
C07930=1195.846,30.366,-45.542,-179.505,5.727,148.866
C07931=1195.851,30.117,-45.527,-179.507,5.726,148.866
C07932=1195.856,29.866,-45.512,-179.510,5.726,148.867
C07933=1195.860,29.617,-45.497,-179.512,5.725,148.868
C07934=1195.866,29.368,-45.481,-179.515,5.725,148.868
C07935=1195.871,29.099,-45.465,-179.518,5.723,148.869
C07936=1195.877,28.830,-45.448,-179.521,5.723,148.870
C07937=1195.882,28.561,-45.433,-179.523,5.722,148.870
C07938=1195.888,28.292,-45.416,-179.526,5.721,148.871
C07939=1195.892,28.043,-45.401,-179.528,5.721,148.872
C07940=1195.898,27.794,-45.386,-179.531,5.720,148.872
C07941=1195.903,27.544,-45.371,-179.533,5.720,148.873
C07942=1195.908,27.295,-45.356,-179.536,5.719,148.873
C07943=1195.913,27.046,-45.341,-179.538,5.718,148.874
C07944=1195.917,26.796,-45.325,-179.541,5.718,148.875
C07945=1195.922,26.546,-45.311,-179.544,5.717,148.875
C07946=1195.928,26.296,-45.295,-179.546,5.717,148.876
C07947=1195.933,26.047,-45.281,-179.548,5.716,148.877
C07948=1195.937,25.798,-45.266,-179.551,5.715,148.877
C07949=1195.943,25.548,-45.250,-179.554,5.715,148.878
C07950=1195.948,25.299,-45.236,-179.556,5.714,148.879
C07951=1195.953,25.049,-45.220,-179.559,5.713,148.879
C07952=1195.958,24.800,-45.205,-179.562,5.712,148.880
C07953=1195.963,24.550,-45.191,-179.564,5.712,148.880
C07954=1195.968,24.301,-45.175,-179.567,5.711,148.881
C07955=1195.973,24.051,-45.161,-179.569,5.710,148.882
C07956=1195.978,23.802,-45.146,-179.572,5.710,148.882
C07957=1195.983,23.552,-45.131,-179.574,5.709,148.883
C07958=1195.988,23.303,-45.116,-179.577,5.709,148.884
C07959=1195.993,23.054,-45.101,-179.579,5.708,148.884
C07960=1195.998,22.804,-45.086,-179.582,5.707,148.885
C07961=1196.002,22.554,-45.071,-179.585,5.707,148.885
C07962=1196.007,22.304,-45.057,-179.587,5.706,148.886
C07963=1196.013,22.055,-45.041,-179.589,5.706,148.887
C07964=1196.018,21.805,-45.027,-179.592,5.705,148.887
C07965=1196.022,21.556,-45.012,-179.595,5.705,148.888
C07966=1196.028,21.306,-44.997,-179.597,5.704,148.889
C07967=1196.033,21.057,-44.982,-179.599,5.703,148.889
C07968=1196.038,20.807,-44.968,-179.602,5.703,148.890
C07969=1196.043,20.557,-44.953,-179.605,5.702,148.890
C07970=1196.048,20.308,-44.938,-179.607,5.702,148.891
C07971=1196.053,20.059,-44.924,-179.610,5.701,148.892
C07972=1196.058,19.809,-44.909,-179.612,5.700,148.892
C07973=1196.064,19.560,-44.894,-179.615,5.700,148.893
C07974=1196.068,19.311,-44.879,-179.617,5.699,148.894
C07975=1196.073,19.061,-44.865,-179.620,5.699,148.894
C07976=1196.078,18.812,-44.851,-179.622,5.698,148.895
C07977=1196.084,18.562,-44.835,-179.625,5.697,148.895
C07978=1196.089,18.313,-44.821,-179.628,5.697,148.896
C07979=1196.093,18.063,-44.806,-179.630,5.696,148.897
C07980=1196.098,17.814,-44.791,-179.632,5.696,148.897
C07981=1196.104,17.564,-44.777,-179.634,5.696,148.898
C07982=1196.109,17.315,-44.762,-179.637,5.695,148.899
C07983=1196.114,17.065,-44.747,-179.640,5.695,148.899
C07984=1196.119,16.815,-44.733,-179.642,5.694,148.900
C07985=1196.123,16.566,-44.718,-179.645,5.693,148.900
C07986=1196.129,16.316,-44.703,-179.647,5.693,148.901
C07987=1196.134,16.066,-44.689,-179.650,5.692,148.902
C07988=1196.139,15.817,-44.674,-179.653,5.692,148.902
C07989=1196.143,15.568,-44.660,-179.655,5.691,148.903
C07990=1196.148,15.318,-44.645,-179.657,5.691,148.904
C07991=1196.154,15.069,-44.631,-179.660,5.690,148.904
C07992=1196.159,14.819,-44.616,-179.663,5.690,148.905
C07993=1196.164,14.570,-44.602,-179.665,5.689,148.906
C07994=1196.169,14.320,-44.587,-179.667,5.688,148.906
C07995=1196.174,14.070,-44.573,-179.670,5.688,148.907
C07996=1196.179,13.821,-44.558,-179.673,5.687,148.907
C07997=1196.184,13.571,-44.544,-179.675,5.687,148.908
C07998=1196.189,13.322,-44.530,-179.678,5.686,148.909
C07999=1196.194,13.072,-44.515,-179.680,5.685,148.909
C08000=1196.200,12.823,-44.500,-179.683,5.685,148.910
C08001=1196.205,12.574,-44.486,-179.686,5.684,148.911
C08002=1196.210,12.324,-44.471,-179.688,5.684,148.911
C08003=1196.215,12.074,-44.457,-179.690,5.683,148.912
C08004=1196.220,11.825,-44.443,-179.693,5.682,148.912
C08005=1196.224,11.575,-44.429,-179.696,5.682,148.913
C08006=1196.229,11.326,-44.414,-179.698,5.681,148.914
C08007=1196.235,11.077,-44.400,-179.700,5.681,148.914
C08008=1196.240,10.827,-44.385,-179.702,5.681,148.915
C08009=1196.245,10.577,-44.371,-179.705,5.680,148.916
C08010=1196.250,10.328,-44.357,-179.708,5.680,148.916
C08011=1196.255,10.078,-44.343,-179.710,5.679,148.917
C08012=1196.259,9.828,-44.328,-179.713,5.679,148.917
C08013=1196.265,9.579,-44.314,-179.715,5.678,148.918
C08014=1196.270,9.329,-44.300,-179.718,5.678,148.919
C08015=1196.275,9.080,-44.285,-179.721,5.677,148.920
C08016=1196.280,8.831,-44.271,-179.723,5.677,148.920
C08017=1196.285,8.581,-44.257,-179.725,5.676,148.921
C08018=1196.289,8.331,-44.242,-179.728,5.675,148.921
C08019=1196.295,8.082,-44.228,-179.731,5.675,148.922
C08020=1196.300,7.832,-44.214,-179.733,5.674,148.923
C08021=1196.305,7.583,-44.200,-179.736,5.674,148.923
C08022=1196.310,7.333,-44.186,-179.738,5.673,148.924
C08023=1196.315,7.083,-44.171,-179.741,5.672,148.925
C08024=1196.320,6.834,-44.157,-179.743,5.673,148.925
C08025=1196.325,6.585,-44.143,-179.746,5.672,148.926
C08026=1196.330,6.335,-44.129,-179.748,5.671,148.926
C08027=1196.335,6.085,-44.115,-179.750,5.671,148.927
C08028=1196.341,5.836,-44.101,-179.753,5.670,148.928
C08029=1196.346,5.587,-44.086,-179.756,5.670,148.928
C08030=1196.351,5.337,-44.072,-179.758,5.669,148.929
C08031=1196.356,5.087,-44.058,-179.760,5.669,148.930
C08032=1196.361,4.838,-44.044,-179.763,5.668,148.930
C08033=1196.366,4.588,-44.030,-179.766,5.668,148.931
C08034=1196.371,4.338,-44.016,-179.768,5.667,148.932
C08035=1196.376,4.088,-44.002,-179.771,5.667,148.932
C08036=1196.381,3.840,-43.988,-179.773,5.666,148.933
C08037=1196.386,3.590,-43.974,-179.775,5.666,148.933
C08038=1196.391,3.340,-43.960,-179.778,5.666,148.934
C08039=1196.397,3.071,-43.945,-179.781,5.665,148.935
C08040=1196.402,2.802,-43.929,-179.783,5.665,148.936
C08041=1196.408,2.533,-43.915,-179.787,5.663,148.936
C08042=1196.413,2.264,-43.900,-179.789,5.663,148.937
C08043=1196.418,2.014,-43.885,-179.791,5.663,148.938
C08044=1196.423,1.764,-43.871,-179.794,5.663,148.938
C08045=1196.429,1.515,-43.857,-179.796,5.662,148.939
C08046=1196.434,1.265,-43.844,-179.799,5.661,148.939
C08047=1196.438,1.016,-43.830,-179.801,5.661,148.940
C08048=1196.444,0.767,-43.816,-179.804,5.660,148.941
C08049=1196.449,0.517,-43.802,-179.807,5.660,148.941
C08050=1196.454,0.267,-43.787,-179.809,5.659,148.942
C08051=1196.459,0.018,-43.774,-179.811,5.658,148.943
C08052=1196.464,-0.232,-43.760,-179.814,5.658,148.943
C08053=1196.469,-0.481,-43.746,-179.816,5.658,148.944
C08054=1196.474,-0.730,-43.732,-179.819,5.658,148.945
C08055=1196.479,-0.981,-43.719,-179.821,5.657,148.945
C08056=1196.484,-1.231,-43.705,-179.824,5.656,148.946
C08057=1196.490,-1.480,-43.691,-179.826,5.656,148.947
C08058=1196.494,-1.729,-43.677,-179.829,5.655,148.947
C08059=1196.499,-1.979,-43.663,-179.832,5.655,148.948
C08060=1196.505,-2.228,-43.649,-179.834,5.654,148.948
C08061=1196.510,-2.478,-43.635,-179.836,5.654,148.949
C08062=1196.514,-2.728,-43.622,-179.839,5.654,148.950
C08063=1196.520,-2.977,-43.608,-179.841,5.653,148.950
C08064=1196.525,-3.227,-43.594,-179.844,5.653,148.951
C08065=1196.531,-3.476,-43.581,-179.846,5.652,148.952
C08066=1196.535,-3.726,-43.567,-179.849,5.652,148.952
C08067=1196.540,-3.975,-43.553,-179.851,5.651,148.953
C08068=1196.546,-4.225,-43.540,-179.854,5.651,148.954
C08069=1196.550,-4.474,-43.526,-179.857,5.650,148.954
C08070=1196.555,-4.724,-43.512,-179.859,5.650,148.955
C08071=1196.561,-4.974,-43.499,-179.861,5.650,148.956
C08072=1196.566,-5.224,-43.484,-179.864,5.649,148.956
C08073=1196.571,-5.472,-43.471,-179.866,5.649,148.957
C08074=1196.576,-5.723,-43.457,-179.869,5.648,148.958
C08075=1196.581,-5.972,-43.443,-179.871,5.648,148.958
C08076=1196.586,-6.222,-43.430,-179.874,5.647,148.959
C08077=1196.591,-6.471,-43.416,-179.876,5.646,148.959
C08078=1196.597,-6.721,-43.403,-179.878,5.647,148.960
C08079=1196.601,-6.970,-43.389,-179.881,5.646,148.961
C08080=1196.607,-7.219,-43.375,-179.884,5.646,148.962
C08081=1196.611,-7.469,-43.362,-179.886,5.645,148.962
C08082=1196.616,-7.719,-43.348,-179.889,5.644,148.963
C08083=1196.622,-7.969,-43.335,-179.891,5.644,148.963
C08084=1196.626,-8.218,-43.321,-179.894,5.643,148.964
C08085=1196.632,-8.468,-43.308,-179.896,5.644,148.965
C08086=1196.637,-8.717,-43.294,-179.898,5.643,148.965
C08087=1196.642,-8.967,-43.281,-179.901,5.642,148.966
C08088=1196.647,-9.216,-43.267,-179.903,5.642,148.967
C08089=1196.652,-9.466,-43.254,-179.906,5.641,148.967
C08090=1196.657,-9.715,-43.240,-179.909,5.641,148.968
C08091=1196.662,-9.966,-43.227,-179.911,5.640,148.968
C08092=1196.667,-10.215,-43.213,-179.913,5.640,148.969
C08093=1196.672,-10.465,-43.200,-179.916,5.640,148.970
C08094=1196.678,-10.714,-43.187,-179.918,5.639,148.971
C08095=1196.683,-10.964,-43.173,-179.921,5.639,148.971
C08096=1196.688,-11.213,-43.160,-179.924,5.639,148.972
C08097=1196.693,-11.463,-43.146,-179.926,5.638,148.972
C08098=1196.698,-11.712,-43.133,-179.928,5.637,148.973
C08099=1196.703,-11.962,-43.119,-179.930,5.638,148.974
C08100=1196.708,-12.211,-43.106,-179.933,5.637,148.974
C08101=1196.713,-12.462,-43.093,-179.936,5.637,148.975
C08102=1196.719,-12.711,-43.079,-179.938,5.636,148.976
C08103=1196.723,-12.961,-43.066,-179.941,5.635,148.976
C08104=1196.729,-13.210,-43.053,-179.943,5.635,148.977
C08105=1196.733,-13.460,-43.039,-179.945,5.635,148.978
C08106=1196.739,-13.709,-43.026,-179.948,5.635,148.978
C08107=1196.744,-13.959,-43.013,-179.950,5.634,148.979
C08108=1196.749,-14.208,-42.999,-179.953,5.633,148.980
C08109=1196.754,-14.458,-42.986,-179.955,5.633,148.980
C08110=1196.760,-14.708,-42.973,-179.958,5.632,148.981
C08111=1196.764,-14.957,-42.960,-179.960,5.633,148.982
C08112=1196.769,-15.207,-42.947,-179.963,5.632,148.982
C08113=1196.775,-15.456,-42.933,-179.965,5.631,148.983
C08114=1196.779,-15.706,-42.920,-179.968,5.631,148.983
C08115=1196.785,-15.955,-42.906,-179.970,5.630,148.984
C08116=1196.789,-16.205,-42.894,-179.973,5.630,148.985
C08117=1196.795,-16.455,-42.880,-179.975,5.630,148.986
C08118=1196.800,-16.704,-42.867,-179.977,5.629,148.986
C08119=1196.805,-16.954,-42.853,-179.980,5.629,148.987
C08120=1196.810,-17.203,-42.841,-179.983,5.628,148.987
C08121=1196.815,-17.453,-42.828,-179.985,5.628,148.988
C08122=1196.821,-17.702,-42.814,-179.987,5.628,148.989
C08123=1196.825,-17.952,-42.801,-179.990,5.628,148.989
C08124=1196.831,-18.202,-42.788,-179.992,5.627,148.990
C08125=1196.836,-18.451,-42.775,-179.995,5.627,148.991
C08126=1196.841,-18.701,-42.762,-179.997,5.626,148.991
C08127=1196.846,-18.950,-42.748,180.000,5.626,148.992
C08128=1196.851,-19.200,-42.735,179.998,5.626,148.993
C08129=1196.857,-19.450,-42.722,179.996,5.625,148.993
C08130=1196.862,-19.699,-42.710,179.993,5.625,148.994
C08131=1196.866,-19.949,-42.697,179.990,5.624,148.995
C08132=1196.872,-20.199,-42.683,179.988,5.624,148.995
C08133=1196.877,-20.448,-42.671,179.986,5.624,148.996
C08134=1196.881,-20.698,-42.657,179.983,5.623,148.996
C08135=1196.887,-20.947,-42.644,179.981,5.623,148.997
C08136=1196.892,-21.197,-42.631,179.978,5.622,148.998
C08137=1196.897,-21.447,-42.618,179.975,5.622,148.999
C08138=1196.903,-21.696,-42.605,179.973,5.622,148.999
C08139=1196.907,-21.946,-42.592,179.971,5.622,149.000
C08140=1196.912,-22.196,-42.580,179.969,5.621,149.000
C08141=1196.918,-22.445,-42.566,179.966,5.620,149.001
C08142=1196.923,-22.695,-42.553,179.963,5.620,149.002
C08143=1196.929,-22.965,-42.540,179.961,5.620,149.002
C08144=1196.934,-23.234,-42.525,179.958,5.620,149.003
C08145=1196.940,-23.504,-42.511,179.956,5.619,149.004
C08146=1196.945,-23.773,-42.498,179.953,5.619,149.005
C08147=1196.950,-24.023,-42.485,179.950,5.618,149.005
C08148=1196.956,-24.272,-42.471,179.948,5.618,149.006
C08149=1196.961,-24.522,-42.459,179.945,5.617,149.007
C08150=1196.965,-24.772,-42.446,179.944,5.617,149.007
C08151=1196.970,-25.021,-42.433,179.941,5.617,149.008
C08152=1196.976,-25.271,-42.420,179.938,5.616,149.008
C08153=1196.981,-25.521,-42.407,179.936,5.616,149.009
C08154=1196.986,-25.770,-42.394,179.933,5.615,149.010
C08155=1196.991,-26.019,-42.382,179.931,5.616,149.011
C08156=1196.997,-26.269,-42.369,179.929,5.615,149.011
C08157=1197.001,-26.519,-42.356,179.926,5.614,149.012
C08158=1197.006,-26.768,-42.343,179.923,5.614,149.012
C08159=1197.012,-27.018,-42.330,179.921,5.614,149.013
C08160=1197.016,-27.268,-42.318,179.919,5.614,149.014
C08161=1197.022,-27.518,-42.305,179.916,5.613,149.014
C08162=1197.027,-27.767,-42.292,179.914,5.613,149.015
C08163=1197.032,-28.017,-42.280,179.911,5.612,149.016
C08164=1197.037,-28.267,-42.267,179.909,5.612,149.016
C08165=1197.042,-28.516,-42.254,179.906,5.612,149.017
C08166=1197.047,-28.765,-42.242,179.904,5.612,149.018
C08167=1197.053,-29.015,-42.228,179.902,5.611,149.018
C08168=1197.058,-29.265,-42.215,179.899,5.611,149.019
C08169=1197.063,-29.515,-42.204,179.897,5.611,149.020
C08170=1197.068,-29.764,-42.191,179.894,5.610,149.020
C08171=1197.073,-30.013,-42.178,179.891,5.610,149.021
C08172=1197.078,-30.263,-42.165,179.890,5.610,149.022
C08173=1197.083,-30.513,-42.153,179.887,5.609,149.022
C08174=1197.089,-30.762,-42.140,179.885,5.609,149.023
C08175=1197.094,-31.012,-42.128,179.882,5.608,149.024
C08176=1197.099,-31.262,-42.115,179.879,5.608,149.024
C08177=1197.104,-31.512,-42.102,179.877,5.608,149.025
C08178=1197.109,-31.761,-42.090,179.875,5.607,149.025
C08179=1197.114,-32.010,-42.077,179.872,5.607,149.026
C08180=1197.120,-32.260,-42.065,179.870,5.606,149.027
C08181=1197.124,-32.510,-42.052,179.868,5.607,149.028
C08182=1197.129,-32.760,-42.040,179.865,5.606,149.028
C08183=1197.134,-33.009,-42.027,179.863,5.605,149.029
C08184=1197.141,-33.259,-42.014,179.860,5.605,149.029
C08185=1197.146,-33.508,-42.002,179.858,5.605,149.030
C08186=1197.150,-33.758,-41.989,179.855,5.605,149.031
C08187=1197.155,-34.008,-41.976,179.853,5.604,149.032
C08188=1197.161,-34.258,-41.964,179.851,5.603,149.032
C08189=1197.166,-34.507,-41.952,179.848,5.604,149.033
C08190=1197.171,-34.756,-41.939,179.846,5.603,149.033
C08191=1197.176,-35.006,-41.927,179.843,5.603,149.034
C08192=1197.181,-35.256,-41.914,179.840,5.602,149.035
C08193=1197.186,-35.506,-41.902,179.838,5.603,149.036
C08194=1197.191,-35.756,-41.890,179.836,5.602,149.036
C08195=1197.197,-36.005,-41.877,179.834,5.601,149.037
C08196=1197.202,-36.254,-41.865,179.831,5.601,149.037
C08197=1197.207,-36.504,-41.853,179.829,5.601,149.038
C08198=1197.212,-36.753,-41.840,179.826,5.601,149.039
C08199=1197.217,-37.003,-41.827,179.824,5.600,149.039
C08200=1197.222,-37.253,-41.815,179.822,5.600,149.040
C08201=1197.227,-37.503,-41.803,179.819,5.600,149.041
C08202=1197.233,-37.753,-41.791,179.817,5.600,149.041
C08203=1197.238,-38.002,-41.778,179.814,5.599,149.042
C08204=1197.243,-38.251,-41.766,179.812,5.599,149.043
C08205=1197.248,-38.501,-41.754,179.810,5.599,149.043
C08206=1197.254,-38.751,-41.741,179.807,5.598,149.044
C08207=1197.259,-39.000,-41.729,179.804,5.598,149.045
C08208=1197.264,-39.250,-41.716,179.802,5.598,149.045
C08209=1197.269,-39.500,-41.704,179.800,5.598,149.046
C08210=1197.274,-39.750,-41.692,179.797,5.597,149.046
C08211=1197.279,-39.999,-41.679,179.795,5.597,149.047
C08212=1197.284,-40.249,-41.668,179.793,5.597,149.048
C08213=1197.289,-40.498,-41.655,179.790,5.596,149.049
C08214=1197.294,-40.748,-41.643,179.787,5.596,149.049
C08215=1197.300,-40.997,-41.631,179.786,5.596,149.050
C08216=1197.305,-41.247,-41.619,179.783,5.595,149.050
C08217=1197.310,-41.496,-41.606,179.780,5.595,149.051
C08218=1197.316,-41.746,-41.594,179.778,5.594,149.052
C08219=1197.321,-41.996,-41.582,179.776,5.595,149.053
C08220=1197.326,-42.246,-41.570,179.773,5.594,149.053
C08221=1197.330,-42.496,-41.558,179.771,5.593,149.054
C08222=1197.335,-42.745,-41.546,179.769,5.594,149.054
C08223=1197.341,-42.995,-41.534,179.766,5.593,149.055
C08224=1197.346,-43.245,-41.521,179.763,5.593,149.056
C08225=1197.351,-43.495,-41.509,179.761,5.592,149.057
C08226=1197.356,-43.744,-41.497,179.759,5.592,149.057
C08227=1197.362,-43.994,-41.485,179.756,5.592,149.058
C08228=1197.366,-44.243,-41.473,179.754,5.591,149.058
C08229=1197.372,-44.493,-41.461,179.752,5.592,149.059
C08230=1197.377,-44.743,-41.449,179.749,5.591,149.060
C08231=1197.382,-44.992,-41.436,179.747,5.591,149.060
C08232=1197.388,-45.242,-41.425,179.745,5.591,149.061
C08233=1197.393,-45.492,-41.413,179.742,5.590,149.062
C08234=1197.397,-45.741,-41.401,179.739,5.590,149.062
C08235=1197.403,-45.991,-41.389,179.737,5.590,149.063
C08236=1197.408,-46.240,-41.376,179.735,5.590,149.064
C08237=1197.413,-46.490,-41.364,179.733,5.589,149.064
C08238=1197.419,-46.740,-41.352,179.730,5.589,149.065
C08239=1197.423,-46.989,-41.340,179.728,5.589,149.066
C08240=1197.429,-47.239,-41.329,179.725,5.588,149.066
C08241=1197.434,-47.489,-41.317,179.722,5.588,149.067
C08242=1197.439,-47.738,-41.304,179.721,5.588,149.068
C08243=1197.444,-47.988,-41.293,179.718,5.588,149.068
C08244=1197.449,-48.238,-41.281,179.716,5.587,149.069
C08245=1197.455,-48.488,-41.269,179.713,5.587,149.070
C08246=1197.460,-48.737,-41.256,179.711,5.587,149.070
C08247=1197.466,-49.007,-41.244,179.708,5.587,149.071
C08248=1197.471,-49.277,-41.231,179.705,5.586,149.072
C08249=1197.476,-49.547,-41.218,179.703,5.586,149.072
C08250=1197.482,-49.817,-41.205,179.700,5.585,149.073
C08251=1197.488,-50.067,-41.193,179.698,5.586,149.074
C08252=1197.492,-50.317,-41.182,179.696,5.585,149.074
C08253=1197.498,-50.566,-41.170,179.693,5.584,149.075
C08254=1197.503,-50.816,-41.158,179.691,5.585,149.076
C08255=1197.508,-51.065,-41.146,179.688,5.584,149.076
C08256=1197.513,-51.315,-41.134,179.686,5.584,149.077
C08257=1197.519,-51.565,-41.123,179.684,5.584,149.078
C08258=1197.524,-51.815,-41.111,179.682,5.583,149.078
C08259=1197.529,-52.065,-41.099,179.679,5.583,149.079
C08260=1197.534,-52.314,-41.087,179.677,5.583,149.080
C08261=1197.539,-52.564,-41.075,179.674,5.583,149.080
C08262=1197.545,-52.813,-41.064,179.672,5.582,149.081
C08263=1197.550,-53.063,-41.052,179.670,5.582,149.082
C08264=1197.555,-53.313,-41.041,179.667,5.582,149.082
C08265=1197.560,-53.563,-41.029,179.665,5.581,149.083
C08266=1197.565,-53.812,-41.016,179.662,5.582,149.084
C08267=1197.570,-54.061,-41.005,179.660,5.581,149.084
C08268=1197.575,-54.311,-40.993,179.658,5.581,149.085
C08269=1197.581,-54.561,-40.981,179.656,5.581,149.086
C08270=1197.585,-54.811,-40.970,179.653,5.580,149.086
C08271=1197.591,-55.061,-40.958,179.650,5.580,149.087
C08272=1197.596,-55.310,-40.947,179.649,5.580,149.088
C08273=1197.602,-55.560,-40.935,179.646,5.580,149.088
C08274=1197.607,-55.810,-40.923,179.643,5.579,149.089
C08275=1197.612,-56.059,-40.912,179.641,5.579,149.090
C08276=1197.617,-56.309,-40.900,179.639,5.579,149.090
C08277=1197.622,-56.558,-40.888,179.636,5.578,149.091
C08278=1197.627,-56.808,-40.876,179.634,5.579,149.092
C08279=1197.632,-57.058,-40.865,179.632,5.578,149.092
C08280=1197.638,-57.307,-40.854,179.629,5.578,149.093
C08281=1197.642,-57.557,-40.842,179.627,5.578,149.094
C08282=1197.648,-57.807,-40.830,179.625,5.577,149.094
C08283=1197.653,-58.057,-40.818,179.622,5.577,149.095
C08284=1197.658,-58.306,-40.807,179.620,5.577,149.096
C08285=1197.663,-58.556,-40.795,179.617,5.577,149.096
C08286=1197.669,-58.805,-40.784,179.615,5.576,149.097
C08287=1197.674,-59.055,-40.772,179.613,5.576,149.097
C08288=1197.679,-59.305,-40.761,179.610,5.576,149.098
C08289=1197.684,-59.555,-40.749,179.608,5.575,149.099
C08290=1197.689,-59.804,-40.738,179.606,5.576,149.100
C08291=1197.695,-60.055,-40.727,179.603,5.575,149.100
C08292=1197.700,-60.304,-40.716,179.601,5.574,149.101
C08293=1197.705,-60.554,-40.704,179.599,5.575,149.101
C08294=1197.710,-60.803,-40.693,179.596,5.574,149.102
C08295=1197.716,-61.053,-40.681,179.593,5.574,149.103
C08296=1197.720,-61.303,-40.670,179.592,5.574,149.103
C08297=1197.726,-61.552,-40.658,179.589,5.573,149.104
C08298=1197.731,-61.802,-40.647,179.586,5.573,149.105
C08299=1197.736,-62.051,-40.635,179.584,5.573,149.105
C08300=1197.741,-62.301,-40.624,179.582,5.573,149.106
C08301=1197.746,-62.551,-40.612,179.580,5.573,149.107
C08302=1197.752,-62.801,-40.601,179.577,5.572,149.107
C08303=1197.757,-63.050,-40.590,179.575,5.572,149.108
C08304=1197.762,-63.300,-40.578,179.573,5.572,149.109
C08305=1197.767,-63.550,-40.567,179.570,5.572,149.109
C08306=1197.773,-63.799,-40.555,179.568,5.571,149.110
C08307=1197.778,-64.049,-40.544,179.566,5.572,149.111
C08308=1197.783,-64.299,-40.534,179.563,5.571,149.111
C08309=1197.788,-64.549,-40.522,179.560,5.571,149.112
C08310=1197.793,-64.798,-40.511,179.559,5.571,149.112
C08311=1197.799,-65.048,-40.499,179.556,5.570,149.113
C08312=1197.803,-65.297,-40.488,179.554,5.571,149.114
C08313=1197.808,-65.547,-40.476,179.551,5.570,149.115
C08314=1197.814,-65.797,-40.466,179.549,5.570,149.115
C08315=1197.819,-66.047,-40.454,179.547,5.570,149.116
C08316=1197.825,-66.296,-40.442,179.544,5.569,149.116
C08317=1197.830,-66.545,-40.431,179.542,5.569,149.117
C08318=1197.835,-66.796,-40.421,179.540,5.569,149.118
C08319=1197.840,-67.046,-40.409,179.537,5.568,149.118
C08320=1197.845,-67.295,-40.398,179.535,5.569,149.119
C08321=1197.850,-67.544,-40.387,179.533,5.568,149.120
C08322=1197.856,-67.795,-40.376,179.530,5.568,149.120
C08323=1197.861,-68.044,-40.364,179.528,5.568,149.121
C08324=1197.866,-68.293,-40.353,179.526,5.567,149.122
C08325=1197.872,-68.544,-40.342,179.523,5.567,149.122
C08326=1197.876,-68.793,-40.331,179.521,5.567,149.123
C08327=1197.882,-69.042,-40.320,179.518,5.567,149.124
C08328=1197.887,-69.293,-40.309,179.517,5.567,149.124
C08329=1197.892,-69.543,-40.298,179.514,5.566,149.125
C08330=1197.897,-69.792,-40.286,179.511,5.566,149.126
C08331=1197.903,-70.042,-40.275,179.509,5.566,149.126
C08332=1197.908,-70.292,-40.264,179.507,5.566,149.127
C08333=1197.913,-70.541,-40.253,179.504,5.565,149.128
C08334=1197.918,-70.791,-40.243,179.502,5.566,149.128
C08335=1197.924,-71.041,-40.231,179.500,5.565,149.129
C08336=1197.929,-71.290,-40.220,179.498,5.565,149.130
C08337=1197.934,-71.540,-40.209,179.495,5.565,149.130
C08338=1197.939,-71.790,-40.197,179.493,5.564,149.131
C08339=1197.945,-72.039,-40.186,179.491,5.565,149.132
C08340=1197.950,-72.289,-40.176,179.488,5.564,149.132
C08341=1197.954,-72.539,-40.165,179.486,5.564,149.133
C08342=1197.961,-72.788,-40.154,179.484,5.564,149.133
C08343=1197.965,-73.038,-40.143,179.481,5.563,149.134
C08344=1197.970,-73.288,-40.132,179.479,5.564,149.135
C08345=1197.976,-73.537,-40.121,179.476,5.563,149.136
C08346=1197.981,-73.787,-40.109,179.475,5.563,149.136
C08347=1197.987,-74.037,-40.099,179.472,5.563,149.137
C08348=1197.991,-74.286,-40.088,179.469,5.562,149.138
C08349=1197.996,-74.537,-40.077,179.467,5.563,149.138
C08350=1198.002,-74.786,-40.066,179.465,5.562,149.139
C08351=1198.007,-75.057,-40.054,179.462,5.561,149.139
C08352=1198.014,-75.327,-40.043,179.460,5.562,149.140
C08353=1198.019,-75.598,-40.030,179.458,5.561,149.141
C08354=1198.024,-75.869,-40.019,179.455,5.561,149.142
C08355=1198.031,-76.119,-40.008,179.453,5.561,149.142
C08356=1198.035,-76.369,-39.997,179.450,5.561,149.143
C08357=1198.040,-76.619,-39.986,179.448,5.561,149.144
C08358=1198.046,-76.868,-39.975,179.446,5.561,149.144
C08359=1198.051,-77.118,-39.965,179.443,5.560,149.145
C08360=1198.056,-77.367,-39.954,179.441,5.560,149.146
C08361=1198.062,-77.617,-39.943,179.439,5.560,149.146
C08362=1198.067,-77.866,-39.932,179.436,5.559,149.147
C08363=1198.072,-78.117,-39.921,179.434,5.560,149.147
C08364=1198.077,-78.366,-39.910,179.432,5.559,149.148
C08365=1198.082,-78.616,-39.900,179.430,5.560,149.149
C08366=1198.087,-78.866,-39.889,179.427,5.559,149.149
C08367=1198.092,-79.115,-39.878,179.425,5.558,149.150
C08368=1198.097,-79.365,-39.867,179.423,5.559,149.151
C08369=1198.104,-79.614,-39.856,179.420,5.558,149.151
C08370=1198.109,-79.865,-39.845,179.418,5.558,149.152
C08371=1198.114,-80.114,-39.835,179.416,5.558,149.153
C08372=1198.119,-80.364,-39.824,179.414,5.558,149.153
C08373=1198.124,-80.613,-39.814,179.411,5.558,149.154
C08374=1198.129,-80.864,-39.803,179.409,5.557,149.155
C08375=1198.135,-81.113,-39.792,179.407,5.557,149.155
C08376=1198.140,-81.363,-39.782,179.404,5.557,149.156
C08377=1198.145,-81.612,-39.771,179.402,5.557,149.157
C08378=1198.150,-81.862,-39.760,179.400,5.557,149.157
C08379=1198.156,-82.112,-39.750,179.398,5.557,149.158
C08380=1198.161,-82.362,-39.739,179.395,5.556,149.159
C08381=1198.166,-82.611,-39.728,179.392,5.556,149.159
C08382=1198.171,-82.861,-39.718,179.391,5.556,149.160
C08383=1198.176,-83.110,-39.708,179.388,5.556,149.161
C08384=1198.181,-83.360,-39.696,179.386,5.556,149.161
C08385=1198.187,-83.610,-39.686,179.383,5.556,149.162
C08386=1198.192,-83.860,-39.675,179.381,5.555,149.162
C08387=1198.198,-84.110,-39.665,179.379,5.555,149.163
C08388=1198.203,-84.359,-39.653,179.376,5.555,149.164
C08389=1198.208,-84.609,-39.643,179.374,5.555,149.165
C08390=1198.213,-84.859,-39.633,179.372,5.554,149.165
C08391=1198.219,-85.109,-39.622,179.370,5.555,149.166
C08392=1198.223,-85.358,-39.612,179.367,5.554,149.166
C08393=1198.229,-85.608,-39.602,179.365,5.554,149.167
C08394=1198.234,-85.858,-39.591,179.363,5.554,149.168
C08395=1198.239,-86.107,-39.581,179.360,5.553,149.168
C08396=1198.244,-86.357,-39.569,179.358,5.554,149.169
C08397=1198.249,-86.607,-39.559,179.356,5.553,149.170
C08398=1198.254,-86.857,-39.549,179.354,5.553,149.170
C08399=1198.260,-87.106,-39.538,179.351,5.553,149.171
C08400=1198.266,-87.356,-39.528,179.349,5.553,149.172
C08401=1198.271,-87.606,-39.518,179.347,5.553,149.172
C08402=1198.276,-87.855,-39.507,179.344,5.552,149.173
C08403=1198.281,-88.105,-39.496,179.342,5.552,149.174
C08404=1198.286,-88.355,-39.486,179.340,5.552,149.174
C08405=1198.291,-88.605,-39.475,179.338,5.552,149.175
C08406=1198.297,-88.855,-39.465,179.335,5.552,149.175
C08407=1198.303,-89.104,-39.455,179.333,5.552,149.176
C08408=1198.307,-89.354,-39.444,179.331,5.552,149.177
C08409=1198.313,-89.603,-39.434,179.329,5.552,149.177
C08410=1198.317,-89.853,-39.424,179.326,5.551,149.178
C08411=1198.323,-90.103,-39.413,179.324,5.551,149.179
C08412=1198.328,-90.352,-39.403,179.322,5.551,149.179
C08413=1198.333,-90.603,-39.393,179.319,5.550,149.180
C08414=1198.339,-90.852,-39.382,179.317,5.551,149.181
C08415=1198.344,-91.102,-39.372,179.315,5.550,149.181
C08416=1198.350,-91.352,-39.362,179.313,5.550,149.182
C08417=1198.355,-91.601,-39.351,179.310,5.550,149.183
C08418=1198.359,-91.851,-39.341,179.308,5.550,149.183
C08419=1198.365,-92.101,-39.331,179.306,5.549,149.184
C08420=1198.370,-92.351,-39.321,179.303,5.549,149.185
C08421=1198.376,-92.601,-39.310,179.301,5.549,149.185
C08422=1198.381,-92.850,-39.299,179.299,5.549,149.186
C08423=1198.386,-93.100,-39.289,179.297,5.549,149.186
C08424=1198.392,-93.349,-39.279,179.294,5.549,149.187
C08425=1198.396,-93.599,-39.269,179.292,5.549,149.188
C08426=1198.401,-93.849,-39.258,179.290,5.548,149.188
C08427=1198.407,-94.098,-39.248,179.288,5.549,149.189
C08428=1198.413,-94.348,-39.238,179.285,5.548,149.190
C08429=1198.418,-94.598,-39.227,179.283,5.549,149.190
C08430=1198.423,-94.848,-39.219,179.281,5.548,149.191
C08431=1198.428,-95.098,-39.208,179.278,5.547,149.192
C08432=1198.433,-95.348,-39.198,179.276,5.548,149.192
C08433=1198.439,-95.597,-39.188,179.274,5.547,149.193
C08434=1198.445,-95.847,-39.177,179.272,5.547,149.194
C08435=1198.449,-96.097,-39.167,179.269,5.547,149.194
C08436=1198.454,-96.346,-39.157,179.268,5.547,149.195
C08437=1198.460,-96.596,-39.147,179.265,5.546,149.195
C08438=1198.465,-96.846,-39.136,179.263,5.547,149.196
C08439=1198.470,-97.095,-39.127,179.260,5.546,149.197
C08440=1198.475,-97.345,-39.117,179.259,5.546,149.197
C08441=1198.480,-97.595,-39.106,179.256,5.546,149.198
C08442=1198.486,-97.845,-39.096,179.254,5.546,149.199
C08443=1198.491,-98.094,-39.086,179.252,5.546,149.199
C08444=1198.497,-98.344,-39.077,179.249,5.545,149.200
C08445=1198.502,-98.594,-39.066,179.247,5.546,149.201
C08446=1198.507,-98.844,-39.056,179.245,5.545,149.201
C08447=1198.512,-99.093,-39.046,179.243,5.545,149.202
C08448=1198.517,-99.343,-39.036,179.240,5.545,149.203
C08449=1198.523,-99.593,-39.026,179.238,5.545,149.203
C08450=1198.528,-99.843,-39.015,179.236,5.544,149.204
C08451=1198.534,-100.092,-39.006,179.234,5.545,149.205
C08452=1198.539,-100.343,-38.996,179.231,5.544,149.205
C08453=1198.544,-100.592,-38.986,179.229,5.544,149.206
C08454=1198.549,-100.841,-38.976,179.227,5.544,149.206
C08455=1198.555,-101.114,-38.965,179.225,5.544,149.207
C08456=1198.561,-101.385,-38.954,179.222,5.544,149.208
C08457=1198.566,-101.656,-38.944,179.219,5.544,149.209
C08458=1198.573,-101.928,-38.933,179.217,5.544,149.209
C08459=1198.577,-102.177,-38.923,179.215,5.543,149.210
C08460=1198.582,-102.427,-38.913,179.213,5.544,149.210
C08461=1198.588,-102.677,-38.902,179.210,5.543,149.211
C08462=1198.593,-102.926,-38.893,179.209,5.543,149.212
C08463=1198.599,-103.176,-38.883,179.206,5.543,149.212
C08464=1198.604,-103.426,-38.873,179.203,5.542,149.213
C08465=1198.609,-103.676,-38.863,179.202,5.542,149.214
C08466=1198.614,-103.925,-38.853,179.199,5.542,149.214
C08467=1198.619,-104.175,-38.844,179.197,5.542,149.215
C08468=1198.625,-104.425,-38.834,179.195,5.542,149.216
C08469=1198.630,-104.675,-38.823,179.193,5.542,149.216
C08470=1198.635,-104.925,-38.814,179.190,5.542,149.217
C08471=1198.641,-105.174,-38.804,179.188,5.542,149.217
C08472=1198.646,-105.423,-38.795,179.186,5.541,149.218
C08473=1198.652,-105.674,-38.785,179.184,5.541,149.219
C08474=1198.657,-105.924,-38.774,179.181,5.541,149.220
C08475=1198.661,-106.173,-38.765,179.179,5.541,149.220
C08476=1198.667,-106.423,-38.755,179.177,5.541,149.221
C08477=1198.672,-106.672,-38.746,179.175,5.541,149.221
C08478=1198.678,-106.922,-38.736,179.172,5.540,149.222
C08479=1198.682,-107.173,-38.726,179.170,5.541,149.223
C08480=1198.688,-107.422,-38.716,179.168,5.540,149.223
C08481=1198.694,-107.672,-38.706,179.166,5.540,149.224
C08482=1198.699,-107.922,-38.697,179.163,5.540,149.225
C08483=1198.704,-108.171,-38.687,179.162,5.540,149.225
C08484=1198.709,-108.420,-38.677,179.159,5.539,149.226
C08485=1198.714,-108.671,-38.667,179.157,5.540,149.226
C08486=1198.719,-108.920,-38.658,179.155,5.539,149.227
C08487=1198.725,-109.171,-38.648,179.153,5.539,149.228
C08488=1198.730,-109.420,-38.639,179.150,5.539,149.228
C08489=1198.736,-109.670,-38.629,179.148,5.539,149.229
C08490=1198.741,-109.919,-38.619,179.146,5.539,149.230
C08491=1198.746,-110.169,-38.609,179.144,5.539,149.230
C08492=1198.751,-110.419,-38.600,179.141,5.538,149.231
C08493=1198.757,-110.669,-38.590,179.139,5.539,149.232
C08494=1198.762,-110.919,-38.581,179.137,5.538,149.232
C08495=1198.767,-111.168,-38.571,179.135,5.538,149.233
C08496=1198.773,-111.418,-38.562,179.132,5.538,149.233
C08497=1198.778,-111.668,-38.552,179.130,5.538,149.234
C08498=1198.783,-111.917,-38.543,179.128,5.537,149.235
C08499=1198.789,-112.167,-38.532,179.126,5.538,149.235
C08500=1198.793,-112.418,-38.523,179.123,5.537,149.236
C08501=1198.799,-112.667,-38.513,179.122,5.537,149.237
C08502=1198.804,-112.917,-38.504,179.119,5.537,149.237
C08503=1198.810,-113.166,-38.494,179.118,5.537,149.238
C08504=1198.815,-113.416,-38.485,179.115,5.537,149.238
C08505=1198.821,-113.666,-38.475,179.113,5.537,149.239
C08506=1198.826,-113.916,-38.466,179.111,5.536,149.240
C08507=1198.831,-114.165,-38.456,179.108,5.537,149.240
C08508=1198.837,-114.415,-38.447,179.106,5.536,149.241
C08509=1198.841,-114.664,-38.437,179.104,5.536,149.242
C08510=1198.847,-114.915,-38.428,179.102,5.536,149.242
C08511=1198.852,-115.164,-38.419,179.099,5.536,149.243
C08512=1198.857,-115.414,-38.409,179.097,5.536,149.243
C08513=1198.863,-115.664,-38.399,179.095,5.536,149.244
C08514=1198.867,-115.914,-38.390,179.093,5.535,149.245
C08515=1198.873,-116.164,-38.380,179.091,5.536,149.245
C08516=1198.879,-116.414,-38.371,179.088,5.535,149.246
C08517=1198.883,-116.663,-38.362,179.087,5.535,149.247
C08518=1198.889,-116.913,-38.352,179.084,5.535,149.247
C08519=1198.894,-117.162,-38.343,179.082,5.535,149.248
C08520=1198.900,-117.413,-38.333,179.080,5.534,149.249
C08521=1198.905,-117.662,-38.324,179.078,5.535,149.249
C08522=1198.910,-117.912,-38.315,179.075,5.534,149.250
C08523=1198.916,-118.162,-38.305,179.073,5.534,149.250
C08524=1198.921,-118.412,-38.296,179.071,5.535,149.251
C08525=1198.926,-118.661,-38.287,179.069,5.534,149.252
C08526=1198.932,-118.911,-38.277,179.067,5.534,149.252
C08527=1198.937,-119.161,-38.268,179.064,5.534,149.253
C08528=1198.942,-119.410,-38.259,179.063,5.534,149.254
C08529=1198.948,-119.660,-38.249,179.060,5.534,149.254
C08530=1198.953,-119.910,-38.240,179.058,5.534,149.255
C08531=1198.958,-120.159,-38.231,179.056,5.533,149.255
C08532=1198.964,-120.409,-38.221,179.054,5.534,149.256
C08533=1198.969,-120.659,-38.212,179.051,5.533,149.257
C08534=1198.974,-120.909,-38.203,179.049,5.533,149.257
C08535=1198.980,-121.159,-38.193,179.047,5.532,149.258
C08536=1198.985,-121.409,-38.184,179.045,5.533,149.259
C08537=1198.990,-121.658,-38.175,179.042,5.532,149.259
C08538=1198.995,-121.908,-38.166,179.041,5.532,149.260
C08539=1199.001,-122.158,-38.156,179.038,5.532,149.261
C08540=1199.006,-122.408,-38.147,179.036,5.532,149.261
C08541=1199.011,-122.658,-38.138,179.034,5.532,149.262
C08542=1199.016,-122.907,-38.129,179.032,5.532,149.262
C08543=1199.022,-123.157,-38.119,179.029,5.531,149.263
C08544=1199.027,-123.407,-38.110,179.027,5.532,149.264
C08545=1199.032,-123.657,-38.101,179.026,5.532,149.264
C08546=1199.037,-123.906,-38.093,179.023,5.531,149.265
C08547=1199.043,-124.156,-38.082,179.021,5.532,149.266
C08548=1199.048,-124.406,-38.073,179.019,5.531,149.266
C08549=1199.053,-124.656,-38.065,179.017,5.531,149.267
C08550=1199.059,-124.906,-38.056,179.015,5.531,149.267
C08551=1199.064,-125.156,-38.046,179.012,5.531,149.268
C08552=1199.069,-125.405,-38.037,179.010,5.531,149.269
C08553=1199.074,-125.655,-38.028,179.008,5.531,149.269
C08554=1199.080,-125.905,-38.019,179.006,5.530,149.270
C08555=1199.085,-126.155,-38.010,179.004,5.530,149.270
C08556=1199.091,-126.405,-38.000,179.001,5.530,149.271
C08557=1199.096,-126.654,-37.992,179.000,5.530,149.272
C08558=1199.102,-126.904,-37.983,178.997,5.529,149.272
C08559=1198.680,-126.914,-38.021,178.994,5.533,149.274
C08560=1198.674,-126.665,-38.029,178.995,5.533,149.274
C08561=1198.669,-126.416,-38.039,178.997,5.533,149.273
C08562=1198.664,-126.166,-38.048,178.999,5.534,149.272
C08563=1198.658,-125.916,-38.058,179.002,5.533,149.272
C08564=1198.653,-125.666,-38.066,179.004,5.534,149.271
C08565=1198.648,-125.416,-38.075,179.006,5.534,149.271
C08566=1198.643,-125.166,-38.084,179.009,5.534,149.270
C08567=1198.637,-124.916,-38.094,179.010,5.534,149.269
C08568=1198.632,-124.667,-38.103,179.013,5.535,149.269
C08569=1198.627,-124.417,-38.112,179.015,5.534,149.268
C08570=1198.622,-124.167,-38.121,179.017,5.535,149.267
C08571=1198.617,-123.917,-38.130,179.019,5.535,149.267
C08572=1198.611,-123.667,-38.139,179.021,5.535,149.266
C08573=1198.606,-123.418,-38.149,179.023,5.535,149.266
C08574=1198.601,-123.168,-38.158,179.026,5.536,149.265
C08575=1198.595,-122.918,-38.167,179.028,5.535,149.264
C08576=1198.590,-122.668,-38.176,179.030,5.536,149.264
C08577=1198.584,-122.418,-38.185,179.032,5.536,149.263
C08578=1198.580,-122.169,-38.195,179.034,5.535,149.262
C08579=1198.574,-121.919,-38.204,179.036,5.536,149.262
C08580=1198.568,-121.669,-38.213,179.038,5.536,149.261
C08581=1198.563,-121.419,-38.222,179.041,5.536,149.260
C08582=1198.558,-121.170,-38.232,179.043,5.536,149.260
C08583=1198.553,-120.920,-38.241,179.045,5.536,149.259
C08584=1198.547,-120.670,-38.250,179.047,5.536,149.259
C08585=1198.543,-120.420,-38.260,179.050,5.537,149.258
C08586=1198.537,-120.170,-38.269,179.052,5.536,149.257
C08587=1198.531,-119.920,-38.278,179.054,5.537,149.257
C08588=1198.526,-119.671,-38.287,179.056,5.537,149.256
C08589=1198.521,-119.421,-38.297,179.058,5.538,149.256
C08590=1198.516,-119.171,-38.306,179.060,5.537,149.255
C08591=1198.510,-118.921,-38.315,179.063,5.538,149.254
C08592=1198.505,-118.672,-38.325,179.065,5.538,149.254
C08593=1198.500,-118.422,-38.334,179.067,5.538,149.253
C08594=1198.494,-118.172,-38.343,179.069,5.538,149.252
C08595=1198.489,-117.923,-38.353,179.072,5.538,149.252
C08596=1198.484,-117.673,-38.362,179.074,5.538,149.251
C08597=1198.478,-117.423,-38.371,179.076,5.539,149.251
C08598=1198.473,-117.173,-38.381,179.078,5.538,149.250
C08599=1198.468,-116.923,-38.390,179.081,5.539,149.249
C08600=1198.463,-116.674,-38.400,179.082,5.539,149.249
C08601=1198.457,-116.424,-38.409,179.084,5.538,149.248
C08602=1198.452,-116.174,-38.418,179.086,5.539,149.248
C08603=1198.447,-115.925,-38.428,179.089,5.539,149.247
C08604=1198.441,-115.675,-38.437,179.091,5.539,149.246
C08605=1198.436,-115.426,-38.447,179.093,5.539,149.246
C08606=1198.430,-115.175,-38.456,179.095,5.539,149.245
C08607=1198.425,-114.926,-38.465,179.098,5.539,149.244
C08608=1198.419,-114.676,-38.476,179.100,5.540,149.244
C08609=1198.414,-114.426,-38.484,179.102,5.539,149.243
C08610=1198.410,-114.176,-38.494,179.105,5.540,149.242
C08611=1198.404,-113.926,-38.504,179.106,5.540,149.242
C08612=1198.399,-113.677,-38.514,179.109,5.540,149.241
C08613=1198.393,-113.427,-38.523,179.110,5.540,149.241
C08614=1198.389,-113.177,-38.533,179.113,5.541,149.240
C08615=1198.383,-112.927,-38.542,179.115,5.540,149.239
C08616=1198.378,-112.678,-38.552,179.117,5.541,149.239
C08617=1198.373,-112.428,-38.561,179.119,5.541,149.238
C08618=1198.367,-112.179,-38.571,179.122,5.541,149.237
C08619=1198.362,-111.929,-38.580,179.124,5.541,149.237
C08620=1198.356,-111.679,-38.590,179.126,5.541,149.236
C08621=1198.352,-111.429,-38.599,179.128,5.541,149.235
C08622=1198.346,-111.179,-38.609,179.131,5.542,149.235
C08623=1198.341,-110.929,-38.618,179.133,5.541,149.234
C08624=1198.335,-110.680,-38.629,179.135,5.542,149.234
C08625=1198.330,-110.430,-38.637,179.137,5.542,149.233
C08626=1198.325,-110.180,-38.648,179.140,5.542,149.232
C08627=1198.319,-109.931,-38.657,179.141,5.542,149.232
C08628=1198.314,-109.680,-38.667,179.144,5.543,149.231
C08629=1198.309,-109.430,-38.676,179.146,5.542,149.230
C08630=1198.304,-109.181,-38.686,179.148,5.543,149.230
C08631=1198.299,-108.932,-38.696,179.150,5.543,149.229
C08632=1198.293,-108.682,-38.705,179.153,5.543,149.228
C08633=1198.288,-108.432,-38.715,179.155,5.543,149.228
C08634=1198.282,-108.182,-38.724,179.157,5.543,149.227
C08635=1198.277,-107.932,-38.735,179.159,5.543,149.226
C08636=1198.272,-107.683,-38.745,179.162,5.544,149.226
C08637=1198.266,-107.432,-38.754,179.164,5.543,149.225
C08638=1198.261,-107.183,-38.764,179.166,5.544,149.225
C08639=1198.256,-106.933,-38.773,179.168,5.544,149.224
C08640=1198.251,-106.684,-38.783,179.171,5.544,149.223
C08641=1198.246,-106.434,-38.793,179.173,5.544,149.223
C08642=1198.241,-106.184,-38.802,179.175,5.545,149.222
C08643=1198.235,-105.934,-38.813,179.177,5.544,149.221
C08644=1198.229,-105.685,-38.823,179.180,5.545,149.221
C08645=1198.224,-105.435,-38.832,179.181,5.545,149.220
C08646=1198.219,-105.185,-38.842,179.184,5.545,149.220
C08647=1198.214,-104.935,-38.852,179.186,5.545,149.219
C08648=1198.209,-104.686,-38.862,179.188,5.545,149.218
C08649=1198.203,-104.436,-38.872,179.191,5.546,149.218
C08650=1198.198,-104.186,-38.881,179.193,5.545,149.217
C08651=1198.193,-103.936,-38.892,179.195,5.546,149.216
C08652=1198.188,-103.686,-38.901,179.197,5.546,149.216
C08653=1198.182,-103.437,-38.911,179.200,5.546,149.215
C08654=1198.177,-103.187,-38.921,179.202,5.546,149.214
C08655=1198.172,-102.937,-38.931,179.204,5.547,149.214
C08656=1198.166,-102.687,-38.940,179.206,5.546,149.213
C08657=1198.161,-102.438,-38.951,179.209,5.547,149.213
C08658=1198.156,-102.188,-38.960,179.211,5.547,149.212
C08659=1198.150,-101.939,-38.971,179.213,5.547,149.211
C08660=1198.145,-101.667,-38.981,179.215,5.547,149.210
C08661=1198.139,-101.395,-38.992,179.218,5.547,149.210
C08662=1198.134,-101.124,-39.003,179.220,5.548,149.209
C08663=1198.128,-100.853,-39.013,179.222,5.548,149.209
C08664=1198.123,-100.603,-39.024,179.225,5.548,149.208
C08665=1198.117,-100.353,-39.034,179.227,5.548,149.207
C08666=1198.112,-100.104,-39.043,179.229,5.548,149.207
C08667=1198.107,-99.854,-39.054,179.231,5.548,149.206
C08668=1198.101,-99.603,-39.064,179.234,5.548,149.205
C08669=1198.096,-99.354,-39.073,179.236,5.548,149.205
C08670=1198.091,-99.105,-39.083,179.238,5.549,149.204
C08671=1198.086,-98.854,-39.094,179.241,5.549,149.203
C08672=1198.080,-98.605,-39.104,179.243,5.549,149.203
C08673=1198.075,-98.356,-39.114,179.245,5.550,149.202
C08674=1198.070,-98.106,-39.124,179.247,5.549,149.201
C08675=1198.064,-97.855,-39.134,179.250,5.550,149.201
C08676=1198.059,-97.606,-39.144,179.252,5.550,149.200
C08677=1198.054,-97.356,-39.154,179.254,5.550,149.199
C08678=1198.049,-97.106,-39.164,179.256,5.550,149.199
C08679=1198.043,-96.857,-39.174,179.259,5.550,149.198
C08680=1198.038,-96.607,-39.185,179.261,5.550,149.198
C08681=1198.034,-96.357,-39.195,179.263,5.550,149.197
C08682=1198.028,-96.108,-39.205,179.265,5.550,149.196
C08683=1198.022,-95.858,-39.215,179.268,5.551,149.196
C08684=1198.017,-95.608,-39.225,179.270,5.551,149.195
C08685=1198.013,-95.359,-39.235,179.272,5.551,149.194
C08686=1198.007,-95.108,-39.245,179.275,5.552,149.194
C08687=1198.001,-94.859,-39.255,179.277,5.551,149.193
C08688=1197.996,-94.609,-39.266,179.279,5.552,149.192
C08689=1197.990,-94.359,-39.276,179.281,5.552,149.192
C08690=1197.986,-94.110,-39.285,179.284,5.552,149.191
C08691=1197.981,-93.860,-39.296,179.286,5.552,149.190
C08692=1197.975,-93.610,-39.306,179.288,5.552,149.190
C08693=1197.970,-93.360,-39.317,179.290,5.552,149.189
C08694=1197.964,-93.110,-39.327,179.293,5.553,149.189
C08695=1197.959,-92.861,-39.337,179.295,5.552,149.188
C08696=1197.955,-92.611,-39.347,179.297,5.553,149.187
C08697=1197.949,-92.361,-39.357,179.300,5.553,149.187
C08698=1197.943,-92.112,-39.368,179.302,5.553,149.186
C08699=1197.938,-91.861,-39.378,179.304,5.553,149.185
C08700=1197.933,-91.613,-39.389,179.306,5.553,149.185
C08701=1197.927,-91.363,-39.399,179.309,5.554,149.184
C08702=1197.922,-91.113,-39.410,179.311,5.553,149.183
C08703=1197.918,-90.863,-39.419,179.313,5.554,149.183
C08704=1197.913,-90.613,-39.430,179.315,5.554,149.182
C08705=1197.907,-90.364,-39.440,179.318,5.554,149.181
C08706=1197.901,-90.114,-39.450,179.320,5.555,149.181
C08707=1197.896,-89.864,-39.461,179.322,5.555,149.180
C08708=1197.891,-89.614,-39.471,179.325,5.555,149.179
C08709=1197.886,-89.364,-39.482,179.327,5.555,149.179
C08710=1197.880,-89.115,-39.492,179.329,5.556,149.178
C08711=1197.875,-88.866,-39.503,179.331,5.555,149.178
C08712=1197.871,-88.616,-39.513,179.334,5.556,149.177
C08713=1197.865,-88.366,-39.523,179.336,5.555,149.176
C08714=1197.860,-88.116,-39.534,179.338,5.556,149.176
C08715=1197.854,-87.866,-39.544,179.341,5.556,149.175
C08716=1197.849,-87.616,-39.554,179.343,5.556,149.174
C08717=1197.844,-87.367,-39.565,179.345,5.557,149.174
C08718=1197.839,-87.118,-39.576,179.347,5.556,149.173
C08719=1197.834,-86.867,-39.586,179.350,5.557,149.172
C08720=1197.828,-86.618,-39.596,179.352,5.557,149.172
C08721=1197.823,-86.368,-39.607,179.354,5.557,149.171
C08722=1197.817,-86.118,-39.617,179.357,5.558,149.170
C08723=1197.813,-85.868,-39.628,179.359,5.557,149.170
C08724=1197.807,-85.619,-39.639,179.361,5.558,149.169
C08725=1197.802,-85.369,-39.649,179.363,5.558,149.169
C08726=1197.796,-85.119,-39.659,179.366,5.558,149.168
C08727=1197.791,-84.869,-39.670,179.368,5.558,149.167
C08728=1197.786,-84.620,-39.681,179.370,5.558,149.166
C08729=1197.781,-84.370,-39.691,179.372,5.559,149.166
C08730=1197.776,-84.120,-39.702,179.375,5.559,149.165
C08731=1197.770,-83.871,-39.712,179.377,5.559,149.164
C08732=1197.765,-83.621,-39.723,179.379,5.559,149.164
C08733=1197.760,-83.371,-39.733,179.382,5.560,149.163
C08734=1197.755,-83.121,-39.744,179.384,5.559,149.163
C08735=1197.749,-82.872,-39.755,179.386,5.560,149.162
C08736=1197.744,-82.622,-39.765,179.388,5.560,149.161
C08737=1197.739,-82.373,-39.776,179.391,5.560,149.161
C08738=1197.734,-82.123,-39.787,179.393,5.560,149.160
C08739=1197.729,-81.873,-39.797,179.395,5.560,149.159
C08740=1197.724,-81.623,-39.808,179.397,5.561,149.159
C08741=1197.718,-81.374,-39.818,179.400,5.560,149.158
C08742=1197.713,-81.124,-39.829,179.402,5.561,149.157
C08743=1197.708,-80.874,-39.839,179.405,5.561,149.157
C08744=1197.703,-80.625,-39.851,179.406,5.561,149.156
C08745=1197.698,-80.375,-39.861,179.409,5.562,149.155
C08746=1197.692,-80.125,-39.872,179.411,5.561,149.155
C08747=1197.687,-79.875,-39.883,179.414,5.562,149.154
C08748=1197.681,-79.625,-39.894,179.416,5.563,149.154
C08749=1197.676,-79.375,-39.904,179.418,5.562,149.153
C08750=1197.671,-79.126,-39.915,179.421,5.563,149.152
C08751=1197.666,-78.876,-39.926,179.423,5.562,149.151
C08752=1197.661,-78.627,-39.937,179.425,5.563,149.151
C08753=1197.656,-78.377,-39.947,179.427,5.563,149.150
C08754=1197.650,-78.127,-39.957,179.430,5.563,149.150
C08755=1197.645,-77.878,-39.969,179.433,5.564,149.149
C08756=1197.640,-77.627,-39.980,179.434,5.564,149.148
C08757=1197.634,-77.378,-39.991,179.437,5.564,149.148
C08758=1197.629,-77.128,-40.001,179.439,5.564,149.147
C08759=1197.624,-76.879,-40.012,179.442,5.564,149.146
C08760=1197.619,-76.629,-40.023,179.444,5.565,149.146
C08761=1197.614,-76.380,-40.034,179.446,5.564,149.145
C08762=1197.608,-76.129,-40.045,179.449,5.565,149.144
C08763=1197.603,-75.880,-40.055,179.451,5.565,149.144
C08764=1197.597,-75.609,-40.067,179.453,5.565,149.143
C08765=1197.592,-75.338,-40.079,179.456,5.565,149.142
C08766=1197.586,-75.068,-40.091,179.459,5.566,149.141
C08767=1197.580,-74.797,-40.103,179.461,5.565,149.141
C08768=1197.575,-74.547,-40.114,179.463,5.566,149.140
C08769=1197.570,-74.298,-40.125,179.466,5.567,149.140
C08770=1197.565,-74.047,-40.135,179.468,5.566,149.139
C08771=1197.559,-73.798,-40.147,179.470,5.567,149.138
C08772=1197.554,-73.548,-40.157,179.472,5.567,149.138
C08773=1197.549,-73.298,-40.169,179.475,5.567,149.137
C08774=1197.544,-73.049,-40.180,179.477,5.568,149.136
C08775=1197.539,-72.799,-40.190,179.479,5.567,149.136
C08776=1197.533,-72.549,-40.202,179.482,5.568,149.135
C08777=1197.528,-72.300,-40.212,179.484,5.568,149.134
C08778=1197.523,-72.050,-40.224,179.486,5.568,149.134
C08779=1197.518,-71.801,-40.234,179.489,5.569,149.133
C08780=1197.512,-71.551,-40.246,179.491,5.568,149.132
C08781=1197.507,-71.301,-40.257,179.493,5.569,149.132
C08782=1197.502,-71.051,-40.267,179.495,5.569,149.131
C08783=1197.496,-70.802,-40.279,179.498,5.569,149.130
C08784=1197.492,-70.552,-40.290,179.501,5.569,149.130
C08785=1197.486,-70.302,-40.301,179.502,5.569,149.129
C08786=1197.481,-70.053,-40.312,179.505,5.570,149.128
C08787=1197.476,-69.802,-40.323,179.508,5.570,149.128
C08788=1197.470,-69.553,-40.334,179.510,5.570,149.127
C08789=1197.466,-69.304,-40.345,179.512,5.571,149.127
C08790=1197.460,-69.053,-40.356,179.514,5.570,149.126
C08791=1197.455,-68.804,-40.367,179.517,5.571,149.125
C08792=1197.450,-68.555,-40.379,179.519,5.571,149.124
C08793=1197.445,-68.305,-40.390,179.521,5.571,149.124
C08794=1197.439,-68.055,-40.401,179.524,5.572,149.123
C08795=1197.434,-67.805,-40.412,179.526,5.572,149.123
C08796=1197.429,-67.555,-40.424,179.528,5.572,149.122
C08797=1197.424,-67.305,-40.434,179.531,5.572,149.121
C08798=1197.419,-67.056,-40.445,179.533,5.572,149.121
C08799=1197.413,-66.806,-40.457,179.535,5.573,149.120
C08800=1197.408,-66.557,-40.469,179.538,5.573,149.119
C08801=1197.403,-66.307,-40.479,179.540,5.573,149.119
C08802=1197.397,-66.057,-40.491,179.543,5.573,149.118
C08803=1197.393,-65.808,-40.502,179.545,5.574,149.117
C08804=1197.387,-65.558,-40.514,179.547,5.574,149.117
C08805=1197.382,-65.308,-40.524,179.550,5.574,149.116
C08806=1197.377,-65.059,-40.535,179.552,5.574,149.115
C08807=1197.372,-64.809,-40.547,179.554,5.575,149.115
C08808=1197.367,-64.559,-40.558,179.557,5.575,149.114
C08809=1197.361,-64.310,-40.570,179.559,5.575,149.113
C08810=1197.356,-64.059,-40.581,179.561,5.575,149.113
C08811=1197.351,-63.810,-40.592,179.564,5.575,149.112
C08812=1197.346,-63.560,-40.604,179.566,5.575,149.111
C08813=1197.340,-63.311,-40.615,179.568,5.576,149.111
C08814=1197.335,-63.061,-40.627,179.571,5.576,149.110
C08815=1197.330,-62.811,-40.638,179.573,5.576,149.109
C08816=1197.325,-62.562,-40.650,179.575,5.577,149.109
C08817=1197.319,-62.312,-40.660,179.577,5.576,149.108
C08818=1197.315,-62.062,-40.671,179.580,5.577,149.107
C08819=1197.309,-61.812,-40.683,179.583,5.577,149.107
C08820=1197.304,-61.563,-40.694,179.585,5.577,149.106
C08821=1197.299,-61.313,-40.706,179.587,5.578,149.106
C08822=1197.294,-61.064,-40.717,179.589,5.578,149.105
C08823=1197.288,-60.814,-40.729,179.592,5.578,149.104
C08824=1197.284,-60.564,-40.740,179.594,5.578,149.103
C08825=1197.278,-60.314,-40.752,179.597,5.579,149.103
C08826=1197.274,-60.065,-40.764,179.598,5.579,149.102
C08827=1197.267,-59.816,-40.775,179.601,5.579,149.102
C08828=1197.262,-59.565,-40.786,179.604,5.580,149.101
C08829=1197.257,-59.315,-40.798,179.606,5.579,149.100
C08830=1197.252,-59.066,-40.809,179.608,5.580,149.100
C08831=1197.247,-58.816,-40.821,179.611,5.581,149.099
C08832=1197.242,-58.567,-40.832,179.613,5.580,149.098
C08833=1197.236,-58.317,-40.844,179.616,5.581,149.098
C08834=1197.232,-58.067,-40.855,179.618,5.581,149.097
C08835=1197.226,-57.817,-40.867,179.620,5.581,149.096
C08836=1197.221,-57.568,-40.878,179.622,5.581,149.096
C08837=1197.216,-57.318,-40.890,179.625,5.582,149.095
C08838=1197.211,-57.069,-40.901,179.627,5.582,149.094
C08839=1197.205,-56.819,-40.913,179.630,5.582,149.094
C08840=1197.200,-56.569,-40.925,179.632,5.583,149.093
C08841=1197.195,-56.320,-40.937,179.634,5.582,149.092
C08842=1197.190,-56.070,-40.948,179.637,5.583,149.092
C08843=1197.185,-55.820,-40.960,179.639,5.583,149.091
C08844=1197.180,-55.571,-40.972,179.642,5.583,149.090
C08845=1197.175,-55.321,-40.983,179.644,5.584,149.090
C08846=1197.169,-55.072,-40.994,179.646,5.584,149.089
C08847=1197.164,-54.822,-41.006,179.648,5.584,149.088
C08848=1197.159,-54.572,-41.018,179.651,5.584,149.088
C08849=1197.154,-54.322,-41.030,179.654,5.585,149.087
C08850=1197.149,-54.073,-41.041,179.655,5.585,149.087
C08851=1197.143,-53.823,-41.053,179.658,5.585,149.086
C08852=1197.138,-53.573,-41.065,179.661,5.586,149.085
C08853=1197.134,-53.324,-41.077,179.663,5.585,149.084
C08854=1197.128,-53.074,-41.088,179.665,5.586,149.084
C08855=1197.123,-52.824,-41.100,179.668,5.587,149.083
C08856=1197.118,-52.575,-41.111,179.670,5.586,149.083
C08857=1197.112,-52.325,-41.123,179.672,5.587,149.082
C08858=1197.107,-52.075,-41.135,179.675,5.587,149.081
C08859=1197.102,-51.826,-41.147,179.677,5.587,149.080
C08860=1197.097,-51.576,-41.159,179.679,5.588,149.080
C08861=1197.091,-51.326,-41.171,179.682,5.588,149.079
C08862=1197.087,-51.076,-41.182,179.684,5.588,149.079
C08863=1197.081,-50.827,-41.194,179.687,5.588,149.078
C08864=1197.076,-50.577,-41.207,179.689,5.589,149.077
C08865=1197.071,-50.328,-41.218,179.691,5.589,149.077
C08866=1197.066,-50.078,-41.230,179.694,5.589,149.076
C08867=1197.061,-49.828,-41.242,179.696,5.590,149.075
C08868=1197.055,-49.558,-41.254,179.699,5.590,149.075
C08869=1197.049,-49.288,-41.267,179.701,5.590,149.074
C08870=1197.044,-49.017,-41.280,179.704,5.590,149.073
C08871=1197.038,-48.748,-41.293,179.706,5.590,149.072
C08872=1197.033,-48.498,-41.305,179.709,5.591,149.072
C08873=1197.028,-48.248,-41.317,179.711,5.591,149.071
C08874=1197.023,-47.999,-41.329,179.713,5.591,149.071
C08875=1197.018,-47.749,-41.340,179.716,5.592,149.070
C08876=1197.012,-47.500,-41.353,179.719,5.592,149.069
C08877=1197.007,-47.250,-41.365,179.721,5.592,149.068
C08878=1197.002,-47.000,-41.376,179.723,5.592,149.068
C08879=1196.997,-46.750,-41.388,179.726,5.593,149.067
C08880=1196.992,-46.501,-41.401,179.728,5.593,149.067
C08881=1196.986,-46.251,-41.413,179.730,5.593,149.066
C08882=1196.982,-46.002,-41.425,179.733,5.594,149.065
C08883=1196.976,-45.752,-41.436,179.735,5.593,149.064
C08884=1196.971,-45.502,-41.448,179.738,5.594,149.064
C08885=1196.966,-45.253,-41.461,179.740,5.595,149.063
C08886=1196.960,-45.003,-41.473,179.743,5.595,149.063
C08887=1196.955,-44.753,-41.485,179.745,5.595,149.062
C08888=1196.951,-44.504,-41.497,179.747,5.595,149.061
C08889=1196.945,-44.254,-41.509,179.750,5.596,149.061
C08890=1196.940,-44.005,-41.521,179.752,5.596,149.060
C08891=1196.935,-43.755,-41.533,179.754,5.596,149.059
C08892=1196.929,-43.505,-41.545,179.757,5.597,149.059
C08893=1196.924,-43.255,-41.558,179.760,5.597,149.058
C08894=1196.919,-43.006,-41.569,179.762,5.597,149.057
C08895=1196.914,-42.756,-41.581,179.764,5.598,149.057
C08896=1196.909,-42.506,-41.593,179.767,5.598,149.056
C08897=1196.904,-42.257,-41.606,179.769,5.598,149.055
C08898=1196.898,-42.007,-41.618,179.771,5.598,149.055
C08899=1196.894,-41.757,-41.631,179.774,5.599,149.054
C08900=1196.888,-41.507,-41.643,179.776,5.599,149.053
C08901=1196.883,-41.257,-41.655,179.778,5.599,149.053
C08902=1196.879,-41.008,-41.667,179.781,5.600,149.052
C08903=1196.873,-40.758,-41.678,179.783,5.600,149.051
C08904=1196.868,-40.509,-41.691,179.786,5.600,149.051
C08905=1196.863,-40.260,-41.704,179.788,5.600,149.050
C08906=1196.857,-40.010,-41.716,179.790,5.601,149.050
C08907=1196.852,-39.760,-41.728,179.793,5.601,149.049
C08908=1196.847,-39.511,-41.740,179.795,5.601,149.048
C08909=1196.842,-39.261,-41.753,179.798,5.601,149.047
C08910=1196.836,-39.011,-41.765,179.800,5.602,149.047
C08911=1196.832,-38.761,-41.778,179.803,5.603,149.046
C08912=1196.826,-38.511,-41.789,179.805,5.602,149.046
C08913=1196.821,-38.262,-41.802,179.807,5.603,149.045
C08914=1196.816,-38.012,-41.814,179.810,5.603,149.044
C08915=1196.811,-37.763,-41.826,179.812,5.603,149.043
C08916=1196.806,-37.513,-41.839,179.814,5.604,149.043
C08917=1196.800,-37.263,-41.851,179.817,5.604,149.042
C08918=1196.795,-37.014,-41.864,179.820,5.605,149.042
C08919=1196.790,-36.765,-41.876,179.822,5.604,149.041
C08920=1196.785,-36.514,-41.888,179.824,5.605,149.040
C08921=1196.780,-36.265,-41.901,179.827,5.606,149.040
C08922=1196.775,-36.015,-41.913,179.829,5.606,149.039
C08923=1196.769,-35.766,-41.926,179.831,5.606,149.038
C08924=1196.764,-35.516,-41.938,179.834,5.606,149.038
C08925=1196.759,-35.266,-41.950,179.837,5.607,149.037
C08926=1196.754,-35.017,-41.963,179.839,5.607,149.036
C08927=1196.749,-34.767,-41.976,179.841,5.607,149.036
C08928=1196.744,-34.517,-41.987,179.844,5.608,149.035
C08929=1196.739,-34.268,-42.000,179.846,5.608,149.034
C08930=1196.734,-34.018,-42.013,179.849,5.609,149.034
C08931=1196.728,-33.769,-42.025,179.851,5.608,149.033
C08932=1196.723,-33.519,-42.037,179.853,5.609,149.032
C08933=1196.718,-33.269,-42.050,179.856,5.610,149.032
C08934=1196.713,-33.020,-42.063,179.858,5.610,149.031
C08935=1196.708,-32.770,-42.075,179.861,5.610,149.030
C08936=1196.703,-32.521,-42.087,179.863,5.610,149.030
C08937=1196.698,-32.271,-42.100,179.865,5.611,149.029
C08938=1196.693,-32.021,-42.113,179.868,5.611,149.028
C08939=1196.688,-31.772,-42.125,179.870,5.611,149.028
C08940=1196.682,-31.522,-42.138,179.873,5.612,149.027
C08941=1196.677,-31.272,-42.150,179.875,5.612,149.026
C08942=1196.672,-31.023,-42.163,179.878,5.612,149.026
C08943=1196.667,-30.773,-42.176,179.880,5.612,149.025
C08944=1196.662,-30.523,-42.188,179.882,5.613,149.025
C08945=1196.657,-30.274,-42.200,179.885,5.613,149.024
C08946=1196.651,-30.025,-42.213,179.888,5.614,149.023
C08947=1196.647,-29.774,-42.226,179.890,5.614,149.022
C08948=1196.641,-29.525,-42.239,179.892,5.614,149.022
C08949=1196.636,-29.276,-42.252,179.895,5.615,149.021
C08950=1196.631,-29.026,-42.264,179.897,5.615,149.021
C08951=1196.626,-28.776,-42.277,179.900,5.616,149.020
C08952=1196.621,-28.526,-42.289,179.902,5.615,149.019
C08953=1196.616,-28.277,-42.302,179.904,5.616,149.019
C08954=1196.611,-28.028,-42.315,179.907,5.617,149.018
C08955=1196.605,-27.777,-42.328,179.909,5.617,149.017
C08956=1196.600,-27.528,-42.341,179.912,5.617,149.017
C08957=1196.595,-27.279,-42.353,179.914,5.617,149.016
C08958=1196.590,-27.029,-42.366,179.917,5.618,149.015
C08959=1196.585,-26.779,-42.379,179.919,5.619,149.015
C08960=1196.580,-26.530,-42.392,179.922,5.619,149.014
C08961=1196.574,-26.280,-42.404,179.924,5.619,149.013
C08962=1196.570,-26.030,-42.417,179.926,5.619,149.013
C08963=1196.564,-25.780,-42.429,179.929,5.620,149.012
C08964=1196.559,-25.531,-42.443,179.931,5.621,149.012
C08965=1196.553,-25.281,-42.455,179.934,5.621,149.011
C08966=1196.549,-25.031,-42.468,179.936,5.621,149.010
C08967=1196.544,-24.782,-42.481,179.939,5.621,149.009
C08968=1196.539,-24.533,-42.493,179.941,5.622,149.009
C08969=1196.533,-24.283,-42.507,179.944,5.622,149.008
C08970=1196.528,-24.033,-42.520,179.946,5.622,149.008
C08971=1196.523,-23.784,-42.532,179.948,5.623,149.007
C08972=1196.517,-23.514,-42.546,179.951,5.623,149.006
C08973=1196.513,-23.245,-42.561,179.954,5.623,149.005
C08974=1196.506,-22.975,-42.575,179.956,5.624,149.005
C08975=1196.501,-22.706,-42.588,179.959,5.624,149.004
C08976=1196.496,-22.456,-42.602,179.962,5.625,149.003
C08977=1196.491,-22.206,-42.615,179.964,5.625,149.003
C08978=1196.486,-21.957,-42.627,179.966,5.625,149.002
C08979=1196.480,-21.707,-42.640,179.969,5.625,149.001
C08980=1196.476,-21.457,-42.653,179.971,5.626,149.001
C08981=1196.470,-21.208,-42.666,179.974,5.627,149.000
C08982=1196.465,-20.958,-42.679,179.976,5.627,148.999
C08983=1196.460,-20.708,-42.692,179.978,5.627,148.999
C08984=1196.455,-20.459,-42.705,179.981,5.627,148.998
C08985=1196.450,-20.209,-42.719,179.983,5.628,148.998
C08986=1196.445,-19.960,-42.732,179.986,5.629,148.997
C08987=1196.440,-19.710,-42.744,179.989,5.629,148.996
C08988=1196.434,-19.460,-42.758,179.991,5.629,148.995
C08989=1196.429,-19.211,-42.770,179.993,5.629,148.995
C08990=1196.424,-18.961,-42.783,179.996,5.630,148.994
C08991=1196.419,-18.712,-42.797,179.998,5.631,148.994
C08992=1196.414,-18.462,-42.810,-179.999,5.631,148.993
C08993=1196.409,-18.212,-42.823,-179.996,5.632,148.992
C08994=1196.404,-17.963,-42.836,-179.994,5.631,148.992
C08995=1196.399,-17.713,-42.849,-179.992,5.632,148.991
C08996=1196.394,-17.464,-42.863,-179.990,5.633,148.990
C08997=1196.389,-17.214,-42.876,-179.987,5.633,148.990
C08998=1196.383,-16.964,-42.889,-179.984,5.634,148.989
C08999=1196.378,-16.715,-42.902,-179.982,5.633,148.988
C09000=1196.374,-16.465,-42.915,-179.980,5.634,148.988
C09001=1196.368,-16.216,-42.929,-179.977,5.635,148.987
C09002=1196.363,-15.966,-42.941,-179.975,5.635,148.986
C09003=1196.358,-15.716,-42.955,-179.972,5.635,148.986
C09004=1196.353,-15.467,-42.968,-179.969,5.636,148.985
C09005=1196.348,-15.217,-42.982,-179.967,5.636,148.984
C09006=1196.342,-14.968,-42.994,-179.965,5.636,148.984
C09007=1196.337,-14.717,-43.008,-179.962,5.637,148.983
C09008=1196.332,-14.469,-43.021,-179.960,5.637,148.983
C09009=1196.327,-14.218,-43.035,-179.957,5.638,148.982
C09010=1196.322,-13.969,-43.047,-179.954,5.638,148.981
C09011=1196.316,-13.720,-43.061,-179.952,5.638,148.980
C09012=1196.312,-13.470,-43.074,-179.950,5.639,148.980
C09013=1196.306,-13.220,-43.087,-179.948,5.639,148.979
C09014=1196.302,-12.971,-43.101,-179.945,5.640,148.979
C09015=1196.296,-12.721,-43.114,-179.942,5.640,148.978
C09016=1196.292,-12.472,-43.128,-179.940,5.641,148.977
C09017=1196.286,-12.222,-43.141,-179.938,5.641,148.977
C09018=1196.281,-11.972,-43.154,-179.935,5.641,148.976
C09019=1196.276,-11.723,-43.168,-179.933,5.642,148.975
C09020=1196.271,-11.473,-43.181,-179.930,5.642,148.975
C09021=1196.266,-11.224,-43.195,-179.927,5.643,148.974
C09022=1196.261,-10.974,-43.208,-179.925,5.644,148.974
C09023=1196.255,-10.725,-43.221,-179.923,5.643,148.973
C09024=1196.251,-10.475,-43.235,-179.921,5.644,148.972
C09025=1196.245,-10.226,-43.248,-179.918,5.644,148.971
C09026=1196.240,-9.976,-43.262,-179.915,5.645,148.971
C09027=1196.236,-9.726,-43.275,-179.913,5.646,148.970
C09028=1196.230,-9.477,-43.289,-179.910,5.646,148.970
C09029=1196.226,-9.227,-43.302,-179.908,5.647,148.969
C09030=1196.220,-8.978,-43.316,-179.906,5.646,148.968
C09031=1196.215,-8.728,-43.329,-179.903,5.647,148.968
C09032=1196.210,-8.479,-43.343,-179.900,5.647,148.967
C09033=1196.205,-8.229,-43.356,-179.898,5.648,148.966
C09034=1196.200,-7.980,-43.370,-179.896,5.648,148.966
C09035=1196.195,-7.729,-43.383,-179.893,5.649,148.965
C09036=1196.189,-7.480,-43.397,-179.890,5.649,148.964
C09037=1196.185,-7.230,-43.410,-179.888,5.649,148.964
C09038=1196.180,-6.981,-43.424,-179.886,5.650,148.963
C09039=1196.174,-6.731,-43.438,-179.883,5.650,148.962
C09040=1196.170,-6.482,-43.451,-179.881,5.651,148.962
C09041=1196.164,-6.232,-43.464,-179.878,5.651,148.961
C09042=1196.160,-5.983,-43.478,-179.875,5.652,148.960
C09043=1196.155,-5.733,-43.492,-179.873,5.653,148.960
C09044=1196.149,-5.483,-43.506,-179.871,5.653,148.959
C09045=1196.144,-5.234,-43.520,-179.868,5.653,148.959
C09046=1196.139,-4.984,-43.532,-179.866,5.653,148.958
C09047=1196.134,-4.735,-43.547,-179.863,5.654,148.957
C09048=1196.129,-4.485,-43.561,-179.861,5.655,148.957
C09049=1196.124,-4.236,-43.574,-179.858,5.655,148.956
C09050=1196.119,-3.986,-43.588,-179.856,5.656,148.955
C09051=1196.113,-3.737,-43.602,-179.853,5.656,148.955
C09052=1196.109,-3.487,-43.615,-179.850,5.657,148.954
C09053=1196.104,-3.237,-43.629,-179.849,5.657,148.953
C09054=1196.098,-2.988,-43.643,-179.846,5.657,148.953
C09055=1196.093,-2.738,-43.657,-179.843,5.658,148.952
C09056=1196.088,-2.489,-43.670,-179.841,5.658,148.951
C09057=1196.083,-2.239,-43.684,-179.838,5.659,148.951
C09058=1196.078,-1.989,-43.698,-179.836,5.660,148.950
C09059=1196.072,-1.740,-43.712,-179.833,5.660,148.950
C09060=1196.068,-1.491,-43.725,-179.831,5.660,148.949
C09061=1196.063,-1.240,-43.739,-179.828,5.661,148.948
C09062=1196.057,-0.991,-43.753,-179.826,5.661,148.947
C09063=1196.052,-0.742,-43.767,-179.824,5.662,148.947
C09064=1196.047,-0.492,-43.781,-179.821,5.662,148.946
C09065=1196.042,-0.243,-43.794,-179.818,5.662,148.946
C09066=1196.037,0.007,-43.808,-179.816,5.663,148.945
C09067=1196.032,0.257,-43.822,-179.813,5.663,148.944
C09068=1196.027,0.506,-43.836,-179.811,5.664,148.944
C09069=1196.022,0.756,-43.851,-179.808,5.665,148.943
C09070=1196.017,1.006,-43.864,-179.806,5.665,148.942
C09071=1196.012,1.255,-43.878,-179.803,5.666,148.942
C09072=1196.007,1.504,-43.892,-179.801,5.665,148.941
C09073=1196.002,1.754,-43.906,-179.799,5.666,148.941
C09074=1195.997,2.004,-43.920,-179.796,5.667,148.940
C09075=1195.991,2.253,-43.934,-179.793,5.667,148.939
C09076=1195.986,2.522,-43.949,-179.791,5.668,148.939
C09077=1195.980,2.792,-43.964,-179.788,5.668,148.938
C09078=1195.975,3.061,-43.979,-179.786,5.669,148.937
C09079=1195.969,3.330,-43.994,-179.783,5.669,148.936
C09080=1195.964,3.579,-44.008,-179.780,5.670,148.936
C09081=1195.960,3.829,-44.022,-179.778,5.670,148.935
C09082=1195.955,4.079,-44.036,-179.775,5.671,148.935
C09083=1195.949,4.328,-44.050,-179.773,5.672,148.934
C09084=1195.944,4.577,-44.064,-179.770,5.672,148.933
C09085=1195.939,4.827,-44.079,-179.767,5.673,148.933
C09086=1195.934,5.077,-44.093,-179.765,5.673,148.932
C09087=1195.929,5.326,-44.107,-179.763,5.674,148.931
C09088=1195.924,5.575,-44.121,-179.760,5.674,148.931
C09089=1195.919,5.825,-44.135,-179.757,5.675,148.930
C09090=1195.914,6.075,-44.150,-179.755,5.675,148.929
C09091=1195.908,6.324,-44.164,-179.753,5.675,148.929
C09092=1195.903,6.574,-44.178,-179.750,5.676,148.928
C09093=1195.899,6.823,-44.191,-179.748,5.676,148.928
C09094=1195.894,7.073,-44.206,-179.745,5.677,148.927
C09095=1195.889,7.322,-44.220,-179.742,5.677,148.926
C09096=1195.884,7.571,-44.234,-179.740,5.678,148.926
C09097=1195.879,7.821,-44.248,-179.738,5.679,148.925
C09098=1195.874,8.071,-44.263,-179.735,5.679,148.924
C09099=1195.869,8.320,-44.277,-179.732,5.680,148.924
C09100=1195.864,8.570,-44.291,-179.730,5.680,148.923
C09101=1195.858,8.819,-44.305,-179.728,5.681,148.923
C09102=1195.853,9.069,-44.319,-179.725,5.682,148.922
C09103=1195.848,9.319,-44.334,-179.722,5.682,148.921
C09104=1195.844,9.568,-44.348,-179.720,5.683,148.920
C09105=1195.839,9.818,-44.362,-179.717,5.683,148.920
C09106=1195.833,10.067,-44.376,-179.715,5.683,148.919
C09107=1195.828,10.317,-44.390,-179.713,5.684,148.919
C09108=1195.822,10.567,-44.405,-179.710,5.684,148.918
C09109=1195.818,10.816,-44.420,-179.707,5.685,148.917
C09110=1195.813,11.066,-44.434,-179.705,5.686,148.917
C09111=1195.808,11.315,-44.449,-179.703,5.686,148.916
C09112=1195.803,11.565,-44.463,-179.700,5.687,148.915
C09113=1195.797,11.814,-44.477,-179.697,5.687,148.915
C09114=1195.792,12.064,-44.491,-179.695,5.688,148.914
C09115=1195.787,12.313,-44.505,-179.692,5.688,148.914
C09116=1195.783,12.563,-44.520,-179.690,5.689,148.913
C09117=1195.778,12.812,-44.535,-179.687,5.689,148.912
C09118=1195.773,13.062,-44.549,-179.685,5.690,148.912
C09119=1195.768,13.312,-44.563,-179.682,5.691,148.911
C09120=1195.762,13.561,-44.578,-179.680,5.691,148.910
C09121=1195.757,13.810,-44.593,-179.677,5.692,148.910
C09122=1195.752,14.060,-44.607,-179.674,5.692,148.909
C09123=1195.747,14.309,-44.621,-179.672,5.693,148.908
C09124=1195.742,14.559,-44.636,-179.670,5.694,148.908
C09125=1195.737,14.808,-44.651,-179.667,5.694,148.907
C09126=1195.732,15.058,-44.665,-179.664,5.695,148.907
C09127=1195.728,15.308,-44.679,-179.662,5.695,148.906
C09128=1195.722,15.558,-44.694,-179.659,5.696,148.905
C09129=1195.717,15.807,-44.709,-179.657,5.696,148.905
C09130=1195.712,16.056,-44.723,-179.654,5.697,148.904
C09131=1195.707,16.306,-44.737,-179.652,5.697,148.903
C09132=1195.702,16.555,-44.752,-179.649,5.698,148.903
C09133=1195.696,16.805,-44.767,-179.647,5.698,148.902
C09134=1195.691,17.054,-44.781,-179.645,5.699,148.902
C09135=1195.687,17.303,-44.796,-179.642,5.699,148.901
C09136=1195.682,17.553,-44.811,-179.639,5.700,148.900
C09137=1195.677,17.803,-44.825,-179.637,5.700,148.900
C09138=1195.671,18.052,-44.840,-179.635,5.701,148.899
C09139=1195.666,18.302,-44.855,-179.632,5.701,148.898
C09140=1195.662,18.552,-44.869,-179.629,5.702,148.898
C09141=1195.657,18.801,-44.884,-179.627,5.703,148.897
C09142=1195.652,19.050,-44.898,-179.624,5.703,148.897
C09143=1195.647,19.300,-44.914,-179.622,5.704,148.896
C09144=1195.642,19.550,-44.928,-179.619,5.704,148.895
C09145=1195.637,19.799,-44.942,-179.617,5.705,148.894
C09146=1195.631,20.049,-44.958,-179.614,5.706,148.894
